Fanuc TP program (LS listing): 190220_hosenrohr_oV1.ls

/PROG  190220_hosenrohr_oV1
/ATTR
COMMENT	= "19-02-22 10:03:29";
PROG_SIZE	= 0;
DEFAULT_GROUP	= 1, 1, *, *, *;
/APPL
    ARC Welding Equipment: 1, *, *, *, *;
/MN
   1:  CALL HOME_ALL;
   1:  UFRAME_NUM = 1;
   1:  UTOOL_NUM = 3;
   1:  COL GUARD ADJUST 150;
   1:  ! -- Layer/Ebene 27 -- !;
   1:  PR[91] = PR[90];
   1:  PR[GP1:91,1] = PR[GP1:90,1] + -0.402;
   1:  PR[GP1:91,2] = PR[GP1:90,2] + 1.190;
   1:  PR[GP1:91,3] = PR[GP1:90,3] + 16.775;
   1:  !Sicherheitspunkt!;
   1:  PR[92] = PR[91];
   1:  PR[92] = PR[GP1:92,3] + 50;
   1:J PR[92];
   1:  !Schweissanfang anfahren!;
   1:L PR[91] R[100]mm/sec CNT100;
   1:  CALL LASER_DRAHT_START;
   1:  PR[GP1:91,1] = PR[GP1:90,1] + -0.660;
   1:  PR[GP1:91,2] = PR[GP1:90,2] + 1.301;
   1:L PR[91] R[100]mm/sec CNT100;
   1:  PR[GP1:91,1] = PR[GP1:90,1] + -2.989;
   1:  PR[GP1:91,2] = PR[GP1:90,2] + 2.142;
   1:L PR[91] R[100]mm/sec CNT100;
   1:  PR[GP1:91,1] = PR[GP1:90,1] + -5.273;
   1:  PR[GP1:91,2] = PR[GP1:90,2] + 6.132;
   1:L PR[91] R[100]mm/sec CNT100;
   1:  PR[GP1:91,1] = PR[GP1:90,1] + -8.308;
   1:  PR[GP1:91,2] = PR[GP1:90,2] + 15.071;
   1:L PR[91] R[100]mm/sec CNT100;
   1:  PR[GP1:91,1] = PR[GP1:90,1] + -9.096;
   1:  PR[GP1:91,2] = PR[GP1:90,2] + 16.647;
   1:L PR[91] R[100]mm/sec CNT100;
   1:  PR[GP1:91,1] = PR[GP1:90,1] + -15.340;
   1:  PR[GP1:91,2] = PR[GP1:90,2] + 24.664;
   1:L PR[91] R[100]mm/sec CNT100;
   1:  PR[GP1:91,1] = PR[GP1:90,1] + -15.998;
   1:  PR[GP1:91,2] = PR[GP1:90,2] + 25.324;
   1:L PR[91] R[100]mm/sec CNT100;
   1:  PR[GP1:91,1] = PR[GP1:90,1] + -25.382;
   1:  PR[GP1:91,2] = PR[GP1:90,2] + 31.412;
   1:L PR[91] R[100]mm/sec CNT100;
   1:  PR[GP1:91,1] = PR[GP1:90,1] + -36.399;
   1:  PR[GP1:91,2] = PR[GP1:90,2] + 34.262;
   1:L PR[91] R[100]mm/sec CNT100;
   1:  PR[GP1:91,1] = PR[GP1:90,1] + -36.821;
   1:  PR[GP1:91,2] = PR[GP1:90,2] + 34.270;
   1:L PR[91] R[100]mm/sec CNT100;
   1:  PR[GP1:91,1] = PR[GP1:90,1] + -47.006;
   1:  PR[GP1:91,2] = PR[GP1:90,2] + 33.504;
   1:L PR[91] R[100]mm/sec CNT100;
   1:  PR[GP1:91,1] = PR[GP1:90,1] + -47.901;
   1:  PR[GP1:91,2] = PR[GP1:90,2] + 33.351;
   1:L PR[91] R[100]mm/sec CNT100;
   1:  PR[GP1:91,1] = PR[GP1:90,1] + -48.764;
   1:  PR[GP1:91,2] = PR[GP1:90,2] + 33.031;
   1:L PR[91] R[100]mm/sec CNT100;
   1:  PR[GP1:91,1] = PR[GP1:90,1] + -57.526;
   1:  PR[GP1:91,2] = PR[GP1:90,2] + 29.256;
   1:L PR[91] R[100]mm/sec CNT100;
   1:  PR[GP1:91,1] = PR[GP1:90,1] + -58.611;
   1:  PR[GP1:91,2] = PR[GP1:90,2] + 28.601;
   1:L PR[91] R[100]mm/sec CNT100;
   1:  PR[GP1:91,1] = PR[GP1:90,1] + -59.584;
   1:  PR[GP1:91,2] = PR[GP1:90,2] + 27.731;
   1:L PR[91] R[100]mm/sec CNT100;
   1:  PR[GP1:91,1] = PR[GP1:90,1] + -66.238;
   1:  PR[GP1:91,2] = PR[GP1:90,2] + 21.668;
   1:L PR[91] R[100]mm/sec CNT100;
   1:  PR[GP1:91,1] = PR[GP1:90,1] + -67.162;
   1:  PR[GP1:91,2] = PR[GP1:90,2] + 20.463;
   1:L PR[91] R[100]mm/sec CNT100;
   1:  PR[GP1:91,1] = PR[GP1:90,1] + -67.875;
   1:  PR[GP1:91,2] = PR[GP1:90,2] + 19.051;
   1:L PR[91] R[100]mm/sec CNT100;
   1:  PR[GP1:91,1] = PR[GP1:90,1] + -71.993;
   1:  PR[GP1:91,2] = PR[GP1:90,2] + 11.491;
   1:L PR[91] R[100]mm/sec CNT100;
   1:  PR[GP1:91,1] = PR[GP1:90,1] + -72.454;
   1:  PR[GP1:91,2] = PR[GP1:90,2] + 9.892;
   1:L PR[91] R[100]mm/sec CNT100;
   1:  PR[GP1:91,1] = PR[GP1:90,1] + -72.617;
   1:  PR[GP1:91,2] = PR[GP1:90,2] + 8.149;
   1:L PR[91] R[100]mm/sec CNT100;
   1:  PR[GP1:91,1] = PR[GP1:90,1] + -73.992;
   1:  PR[GP1:91,2] = PR[GP1:90,2] + -0.094;
   1:L PR[91] R[100]mm/sec CNT100;
   1:  PR[GP1:91,1] = PR[GP1:90,1] + -73.819;
   1:  PR[GP1:91,2] = PR[GP1:90,2] + -1.941;
   1:L PR[91] R[100]mm/sec CNT100;
   1:  PR[GP1:91,1] = PR[GP1:90,1] + -72.460;
   1:  PR[GP1:91,2] = PR[GP1:90,2] + -10.015;
   1:L PR[91] R[100]mm/sec CNT100;
   1:  PR[GP1:91,1] = PR[GP1:90,1] + -71.991;
   1:  PR[GP1:91,2] = PR[GP1:90,2] + -11.644;
   1:L PR[91] R[100]mm/sec CNT100;
   1:  PR[GP1:91,1] = PR[GP1:90,1] + -71.216;
   1:  PR[GP1:91,2] = PR[GP1:90,2] + -13.179;
   1:L PR[91] R[100]mm/sec CNT100;
   1:  PR[GP1:91,1] = PR[GP1:90,1] + -67.168;
   1:  PR[GP1:91,2] = PR[GP1:90,2] + -20.599;
   1:L PR[91] R[100]mm/sec CNT100;
   1:  PR[GP1:91,1] = PR[GP1:90,1] + -66.239;
   1:  PR[GP1:91,2] = PR[GP1:90,2] + -21.810;
   1:L PR[91] R[100]mm/sec CNT100;
   1:  PR[GP1:91,1] = PR[GP1:90,1] + -65.065;
   1:  PR[GP1:91,2] = PR[GP1:90,2] + -22.860;
   1:L PR[91] R[100]mm/sec CNT100;
   1:  PR[GP1:91,1] = PR[GP1:90,1] + -58.609;
   1:  PR[GP1:91,2] = PR[GP1:90,2] + -28.747;
   1:L PR[91] R[100]mm/sec CNT100;
   1:  PR[GP1:91,1] = PR[GP1:90,1] + -57.539;
   1:  PR[GP1:91,2] = PR[GP1:90,2] + -29.392;
   1:L PR[91] R[100]mm/sec CNT100;
   1:  PR[GP1:91,1] = PR[GP1:90,1] + -56.298;
   1:  PR[GP1:91,2] = PR[GP1:90,2] + -29.853;
   1:L PR[91] R[100]mm/sec CNT100;
   1:  PR[GP1:91,1] = PR[GP1:90,1] + -47.885;
   1:  PR[GP1:91,2] = PR[GP1:90,2] + -33.498;
   1:L PR[91] R[100]mm/sec CNT100;
   1:  PR[GP1:91,1] = PR[GP1:90,1] + -47.006;
   1:  PR[GP1:91,2] = PR[GP1:90,2] + -33.648;
   1:L PR[91] R[100]mm/sec CNT100;
   1:  PR[GP1:91,1] = PR[GP1:90,1] + -36.821;
   1:  PR[GP1:91,2] = PR[GP1:90,2] + -34.414;
   1:L PR[91] R[100]mm/sec CNT100;
   1:  PR[GP1:91,1] = PR[GP1:90,1] + -36.385;
   1:  PR[GP1:91,2] = PR[GP1:90,2] + -34.406;
   1:L PR[91] R[100]mm/sec CNT100;
   1:  PR[GP1:91,1] = PR[GP1:90,1] + -35.945;
   1:  PR[GP1:91,2] = PR[GP1:90,2] + -34.315;
   1:L PR[91] R[100]mm/sec CNT100;
   1:  PR[GP1:91,1] = PR[GP1:90,1] + -25.382;
   1:  PR[GP1:91,2] = PR[GP1:90,2] + -31.557;
   1:L PR[91] R[100]mm/sec CNT100;
   1:  PR[GP1:91,1] = PR[GP1:90,1] + -15.998;
   1:  PR[GP1:91,2] = PR[GP1:90,2] + -25.468;
   1:L PR[91] R[100]mm/sec CNT100;
   1:  PR[GP1:91,1] = PR[GP1:90,1] + -15.340;
   1:  PR[GP1:91,2] = PR[GP1:90,2] + -24.808;
   1:L PR[91] R[100]mm/sec CNT100;
   1:  PR[GP1:91,1] = PR[GP1:90,1] + -9.096;
   1:  PR[GP1:91,2] = PR[GP1:90,2] + -16.791;
   1:L PR[91] R[100]mm/sec CNT100;
   1:  PR[GP1:91,1] = PR[GP1:90,1] + -8.309;
   1:  PR[GP1:91,2] = PR[GP1:90,2] + -15.219;
   1:L PR[91] R[100]mm/sec CNT100;
   1:  PR[GP1:91,1] = PR[GP1:90,1] + -5.290;
   1:  PR[GP1:91,2] = PR[GP1:90,2] + -6.326;
   1:L PR[91] R[100]mm/sec CNT100;
   1:  PR[GP1:91,1] = PR[GP1:90,1] + -4.379;
   1:  PR[GP1:91,2] = PR[GP1:90,2] + -3.772;
   1:L PR[91] R[100]mm/sec CNT100;
   1:  PR[GP1:91,1] = PR[GP1:90,1] + -3.822;
   1:  PR[GP1:91,2] = PR[GP1:90,2] + -3.156;
   1:L PR[91] R[100]mm/sec CNT100;
   1:  PR[GP1:91,1] = PR[GP1:90,1] + -3.023;
   1:  PR[GP1:91,2] = PR[GP1:90,2] + -2.452;
   1:L PR[91] R[100]mm/sec CNT100;
   1:  PR[GP1:91,1] = PR[GP1:90,1] + -2.740;
   1:  PR[GP1:91,2] = PR[GP1:90,2] + -2.161;
   1:L PR[91] R[100]mm/sec CNT100;
   1:  PR[GP1:91,1] = PR[GP1:90,1] + -2.333;
   1:  PR[GP1:91,2] = PR[GP1:90,2] + -1.998;
   1:L PR[91] R[100]mm/sec CNT100;
   1:  PR[GP1:91,1] = PR[GP1:90,1] + -0.802;
   1:  PR[GP1:91,2] = PR[GP1:90,2] + -1.217;
   1:L PR[91] R[100]mm/sec CNT100;
   1:  PR[GP1:91,1] = PR[GP1:90,1] + 0.616;
   1:  PR[GP1:91,2] = PR[GP1:90,2] + -1.334;
   1:L PR[91] R[100]mm/sec CNT100;
   1:  PR[GP1:91,1] = PR[GP1:90,1] + 0.873;
   1:  PR[GP1:91,2] = PR[GP1:90,2] + -1.445;
   1:L PR[91] R[100]mm/sec CNT100;
   1:  PR[GP1:91,1] = PR[GP1:90,1] + 3.204;
   1:  PR[GP1:91,2] = PR[GP1:90,2] + -2.287;
   1:L PR[91] R[100]mm/sec CNT100;
   1:  PR[GP1:91,1] = PR[GP1:90,1] + 3.775;
   1:  PR[GP1:91,2] = PR[GP1:90,2] + -3.292;
   1:L PR[91] R[100]mm/sec CNT100;
   1:  PR[GP1:91,1] = PR[GP1:90,1] + 5.076;
   1:  PR[GP1:91,2] = PR[GP1:90,2] + -5.769;
   1:L PR[91] R[100]mm/sec CNT100;
   1:  PR[GP1:91,1] = PR[GP1:90,1] + 5.465;
   1:  PR[GP1:91,2] = PR[GP1:90,2] + -6.220;
   1:L PR[91] R[100]mm/sec CNT100;
   1:  PR[GP1:91,1] = PR[GP1:90,1] + 8.520;
   1:  PR[GP1:91,2] = PR[GP1:90,2] + -15.214;
   1:L PR[91] R[100]mm/sec CNT100;
   1:  PR[GP1:91,1] = PR[GP1:90,1] + 9.306;
   1:  PR[GP1:91,2] = PR[GP1:90,2] + -16.783;
   1:L PR[91] R[100]mm/sec CNT100;
   1:  PR[GP1:91,1] = PR[GP1:90,1] + 15.550;
   1:  PR[GP1:91,2] = PR[GP1:90,2] + -24.804;
   1:L PR[91] R[100]mm/sec CNT100;
   1:  PR[GP1:91,1] = PR[GP1:90,1] + 16.209;
   1:  PR[GP1:91,2] = PR[GP1:90,2] + -25.466;
   1:L PR[91] R[100]mm/sec CNT100;
   1:  PR[GP1:91,1] = PR[GP1:90,1] + 25.593;
   1:  PR[GP1:91,2] = PR[GP1:90,2] + -31.555;
   1:L PR[91] R[100]mm/sec CNT100;
   1:  PR[GP1:91,1] = PR[GP1:90,1] + 36.611;
   1:  PR[GP1:91,2] = PR[GP1:90,2] + -34.406;
   1:L PR[91] R[100]mm/sec CNT100;
   1:  PR[GP1:91,1] = PR[GP1:90,1] + 37.032;
   1:  PR[GP1:91,2] = PR[GP1:90,2] + -34.414;
   1:L PR[91] R[100]mm/sec CNT100;
   1:  PR[GP1:91,1] = PR[GP1:90,1] + 47.218;
   1:  PR[GP1:91,2] = PR[GP1:90,2] + -33.648;
   1:L PR[91] R[100]mm/sec CNT100;
   1:  PR[GP1:91,1] = PR[GP1:90,1] + 48.113;
   1:  PR[GP1:91,2] = PR[GP1:90,2] + -33.495;
   1:L PR[91] R[100]mm/sec CNT100;
   1:  PR[GP1:91,1] = PR[GP1:90,1] + 48.975;
   1:  PR[GP1:91,2] = PR[GP1:90,2] + -33.175;
   1:L PR[91] R[100]mm/sec CNT100;
   1:  PR[GP1:91,1] = PR[GP1:90,1] + 57.738;
   1:  PR[GP1:91,2] = PR[GP1:90,2] + -29.401;
   1:L PR[91] R[100]mm/sec CNT100;
   1:  PR[GP1:91,1] = PR[GP1:90,1] + 58.824;
   1:  PR[GP1:91,2] = PR[GP1:90,2] + -28.746;
   1:L PR[91] R[100]mm/sec CNT100;
   1:  PR[GP1:91,1] = PR[GP1:90,1] + 59.797;
   1:  PR[GP1:91,2] = PR[GP1:90,2] + -27.876;
   1:L PR[91] R[100]mm/sec CNT100;
   1:  PR[GP1:91,1] = PR[GP1:90,1] + 66.450;
   1:  PR[GP1:91,2] = PR[GP1:90,2] + -21.811;
   1:L PR[91] R[100]mm/sec CNT100;
   1:  PR[GP1:91,1] = PR[GP1:90,1] + 67.375;
   1:  PR[GP1:91,2] = PR[GP1:90,2] + -20.606;
   1:L PR[91] R[100]mm/sec CNT100;
   1:  PR[GP1:91,1] = PR[GP1:90,1] + 68.088;
   1:  PR[GP1:91,2] = PR[GP1:90,2] + -19.193;
   1:L PR[91] R[100]mm/sec CNT100;
   1:  PR[GP1:91,1] = PR[GP1:90,1] + 72.207;
   1:  PR[GP1:91,2] = PR[GP1:90,2] + -11.638;
   1:L PR[91] R[100]mm/sec CNT100;
   1:  PR[GP1:91,1] = PR[GP1:90,1] + 72.667;
   1:  PR[GP1:91,2] = PR[GP1:90,2] + -10.040;
   1:L PR[91] R[100]mm/sec CNT100;
   1:  PR[GP1:91,1] = PR[GP1:90,1] + 72.830;
   1:  PR[GP1:91,2] = PR[GP1:90,2] + -8.297;
   1:L PR[91] R[100]mm/sec CNT100;
   1:  PR[GP1:91,1] = PR[GP1:90,1] + 74.205;
   1:  PR[GP1:91,2] = PR[GP1:90,2] + -0.050;
   1:L PR[91] R[100]mm/sec CNT100;
   1:  PR[GP1:91,1] = PR[GP1:90,1] + 74.032;
   1:  PR[GP1:91,2] = PR[GP1:90,2] + 1.797;
   1:L PR[91] R[100]mm/sec CNT100;
   1:  PR[GP1:91,1] = PR[GP1:90,1] + 72.673;
   1:  PR[GP1:91,2] = PR[GP1:90,2] + 9.874;
   1:L PR[91] R[100]mm/sec CNT100;
   1:  PR[GP1:91,1] = PR[GP1:90,1] + 72.204;
   1:  PR[GP1:91,2] = PR[GP1:90,2] + 11.504;
   1:L PR[91] R[100]mm/sec CNT100;
   1:  PR[GP1:91,1] = PR[GP1:90,1] + 71.429;
   1:  PR[GP1:91,2] = PR[GP1:90,2] + 13.039;
   1:L PR[91] R[100]mm/sec CNT100;
   1:  PR[GP1:91,1] = PR[GP1:90,1] + 67.381;
   1:  PR[GP1:91,2] = PR[GP1:90,2] + 20.454;
   1:L PR[91] R[100]mm/sec CNT100;
   1:  PR[GP1:91,1] = PR[GP1:90,1] + 66.452;
   1:  PR[GP1:91,2] = PR[GP1:90,2] + 21.665;
   1:L PR[91] R[100]mm/sec CNT100;
   1:  PR[GP1:91,1] = PR[GP1:90,1] + 65.278;
   1:  PR[GP1:91,2] = PR[GP1:90,2] + 22.715;
   1:L PR[91] R[100]mm/sec CNT100;
   1:  PR[GP1:91,1] = PR[GP1:90,1] + 58.821;
   1:  PR[GP1:91,2] = PR[GP1:90,2] + 28.604;
   1:L PR[91] R[100]mm/sec CNT100;
   1:  PR[GP1:91,1] = PR[GP1:90,1] + 57.752;
   1:  PR[GP1:91,2] = PR[GP1:90,2] + 29.249;
   1:L PR[91] R[100]mm/sec CNT100;
   1:  PR[GP1:91,1] = PR[GP1:90,1] + 56.510;
   1:  PR[GP1:91,2] = PR[GP1:90,2] + 29.710;
   1:L PR[91] R[100]mm/sec CNT100;
   1:  PR[GP1:91,1] = PR[GP1:90,1] + 48.097;
   1:  PR[GP1:91,2] = PR[GP1:90,2] + 33.354;
   1:L PR[91] R[100]mm/sec CNT100;
   1:  PR[GP1:91,1] = PR[GP1:90,1] + 47.218;
   1:  PR[GP1:91,2] = PR[GP1:90,2] + 33.504;
   1:L PR[91] R[100]mm/sec CNT100;
   1:  PR[GP1:91,1] = PR[GP1:90,1] + 37.032;
   1:  PR[GP1:91,2] = PR[GP1:90,2] + 34.270;
   1:L PR[91] R[100]mm/sec CNT100;
   1:  PR[GP1:91,1] = PR[GP1:90,1] + 36.596;
   1:  PR[GP1:91,2] = PR[GP1:90,2] + 34.262;
   1:L PR[91] R[100]mm/sec CNT100;
   1:  PR[GP1:91,1] = PR[GP1:90,1] + 36.157;
   1:  PR[GP1:91,2] = PR[GP1:90,2] + 34.171;
   1:L PR[91] R[100]mm/sec CNT100;
   1:  PR[GP1:91,1] = PR[GP1:90,1] + 25.593;
   1:  PR[GP1:91,2] = PR[GP1:90,2] + 31.412;
   1:L PR[91] R[100]mm/sec CNT100;
   1:  PR[GP1:91,1] = PR[GP1:90,1] + 16.209;
   1:  PR[GP1:91,2] = PR[GP1:90,2] + 25.322;
   1:L PR[91] R[100]mm/sec CNT100;
   1:  PR[GP1:91,1] = PR[GP1:90,1] + 15.550;
   1:  PR[GP1:91,2] = PR[GP1:90,2] + 24.660;
   1:L PR[91] R[100]mm/sec CNT100;
   1:  PR[GP1:91,1] = PR[GP1:90,1] + 9.306;
   1:  PR[GP1:91,2] = PR[GP1:90,2] + 16.639;
   1:L PR[91] R[100]mm/sec CNT100;
   1:  PR[GP1:91,1] = PR[GP1:90,1] + 8.518;
   1:  PR[GP1:91,2] = PR[GP1:90,2] + 15.066;
   1:L PR[91] R[100]mm/sec CNT100;
   1:  PR[GP1:91,1] = PR[GP1:90,1] + 5.502;
   1:  PR[GP1:91,2] = PR[GP1:90,2] + 6.182;
   1:L PR[91] R[100]mm/sec CNT100;
   1:  PR[GP1:91,1] = PR[GP1:90,1] + 4.592;
   1:  PR[GP1:91,2] = PR[GP1:90,2] + 3.627;
   1:L PR[91] R[100]mm/sec CNT100;
   1:  PR[GP1:91,1] = PR[GP1:90,1] + 4.036;
   1:  PR[GP1:91,2] = PR[GP1:90,2] + 3.013;
   1:L PR[91] R[100]mm/sec CNT100;
   1:  PR[GP1:91,1] = PR[GP1:90,1] + 3.236;
   1:  PR[GP1:91,2] = PR[GP1:90,2] + 2.309;
   1:L PR[91] R[100]mm/sec CNT100;
   1:  PR[GP1:91,1] = PR[GP1:90,1] + 2.954;
   1:  PR[GP1:91,2] = PR[GP1:90,2] + 2.018;
   1:L PR[91] R[100]mm/sec CNT100;
   1:  PR[GP1:91,1] = PR[GP1:90,1] + 2.547;
   1:  PR[GP1:91,2] = PR[GP1:90,2] + 1.854;
   1:L PR[91] R[100]mm/sec CNT100;
   1:  PR[GP1:91,1] = PR[GP1:90,1] + 1.015;
   1:  PR[GP1:91,2] = PR[GP1:90,2] + 1.073;
   1:L PR[91] R[100]mm/sec CNT100;
   1:  ! -- Layer/Ebene 28 -- !;
   1:  PR[91] = PR[90];
   1:  PR[GP1:91,1] = PR[GP1:90,1] + -1.935;
   1:  PR[GP1:91,2] = PR[GP1:90,2] + 1.929;
   1:  PR[GP1:91,3] = PR[GP1:90,3] + 17.385;
   1:L PR[91] R[100]mm/sec CNT100;
   1:  PR[GP1:91,1] = PR[GP1:90,1] + -2.796;
   1:  PR[GP1:91,2] = PR[GP1:90,2] + 2.294;
   1:L PR[91] R[100]mm/sec CNT100;
   1:  PR[GP1:91,1] = PR[GP1:90,1] + -5.248;
   1:  PR[GP1:91,2] = PR[GP1:90,2] + 6.572;
   1:L PR[91] R[100]mm/sec CNT100;
   1:  PR[GP1:91,1] = PR[GP1:90,1] + -7.950;
   1:  PR[GP1:91,2] = PR[GP1:90,2] + 14.528;
   1:L PR[91] R[100]mm/sec CNT100;
   1:  PR[GP1:91,1] = PR[GP1:90,1] + -9.175;
   1:  PR[GP1:91,2] = PR[GP1:90,2] + 16.979;
   1:L PR[91] R[100]mm/sec CNT100;
   1:  PR[GP1:91,1] = PR[GP1:90,1] + -14.817;
   1:  PR[GP1:91,2] = PR[GP1:90,2] + 24.222;
   1:L PR[91] R[100]mm/sec CNT100;
   1:  PR[GP1:91,1] = PR[GP1:90,1] + -16.126;
   1:  PR[GP1:91,2] = PR[GP1:90,2] + 25.535;
   1:L PR[91] R[100]mm/sec CNT100;
   1:  PR[GP1:91,1] = PR[GP1:90,1] + -24.751;
   1:  PR[GP1:91,2] = PR[GP1:90,2] + 31.136;
   1:L PR[91] R[100]mm/sec CNT100;
   1:  PR[GP1:91,1] = PR[GP1:90,1] + -25.479;
   1:  PR[GP1:91,2] = PR[GP1:90,2] + 31.508;
   1:L PR[91] R[100]mm/sec CNT100;
   1:  PR[GP1:91,1] = PR[GP1:90,1] + -34.683;
   1:  PR[GP1:91,2] = PR[GP1:90,2] + 33.823;
   1:L PR[91] R[100]mm/sec CNT100;
   1:  PR[GP1:91,1] = PR[GP1:90,1] + -36.395;
   1:  PR[GP1:91,2] = PR[GP1:90,2] + 34.266;
   1:L PR[91] R[100]mm/sec CNT100;
   1:  PR[GP1:91,1] = PR[GP1:90,1] + -47.334;
   1:  PR[GP1:91,2] = PR[GP1:90,2] + 33.451;
   1:L PR[91] R[100]mm/sec CNT100;
   1:  PR[GP1:91,1] = PR[GP1:90,1] + -47.835;
   1:  PR[GP1:91,2] = PR[GP1:90,2] + 33.366;
   1:L PR[91] R[100]mm/sec CNT100;
   1:  PR[GP1:91,1] = PR[GP1:90,1] + -48.324;
   1:  PR[GP1:91,2] = PR[GP1:90,2] + 33.184;
   1:L PR[91] R[100]mm/sec CNT100;
   1:  PR[GP1:91,1] = PR[GP1:90,1] + -57.721;
   1:  PR[GP1:91,2] = PR[GP1:90,2] + 29.136;
   1:L PR[91] R[100]mm/sec CNT100;
   1:  PR[GP1:91,1] = PR[GP1:90,1] + -58.486;
   1:  PR[GP1:91,2] = PR[GP1:90,2] + 28.675;
   1:L PR[91] R[100]mm/sec CNT100;
   1:  PR[GP1:91,1] = PR[GP1:90,1] + -66.319;
   1:  PR[GP1:91,2] = PR[GP1:90,2] + 21.549;
   1:L PR[91] R[100]mm/sec CNT100;
   1:  PR[GP1:91,1] = PR[GP1:90,1] + -67.028;
   1:  PR[GP1:91,2] = PR[GP1:90,2] + 20.624;
   1:L PR[91] R[100]mm/sec CNT100;
   1:  PR[GP1:91,1] = PR[GP1:90,1] + -67.582;
   1:  PR[GP1:91,2] = PR[GP1:90,2] + 19.527;
   1:L PR[91] R[100]mm/sec CNT100;
   1:  PR[GP1:91,1] = PR[GP1:90,1] + -71.999;
   1:  PR[GP1:91,2] = PR[GP1:90,2] + 11.419;
   1:L PR[91] R[100]mm/sec CNT100;
   1:  PR[GP1:91,1] = PR[GP1:90,1] + -72.365;
   1:  PR[GP1:91,2] = PR[GP1:90,2] + 10.149;
   1:L PR[91] R[100]mm/sec CNT100;
   1:  PR[GP1:91,1] = PR[GP1:90,1] + -72.496;
   1:  PR[GP1:91,2] = PR[GP1:90,2] + 8.747;
   1:L PR[91] R[100]mm/sec CNT100;
   1:  PR[GP1:91,1] = PR[GP1:90,1] + -73.971;
   1:  PR[GP1:91,2] = PR[GP1:90,2] + -0.094;
   1:L PR[91] R[100]mm/sec CNT100;
   1:  PR[GP1:91,1] = PR[GP1:90,1] + -73.828;
   1:  PR[GP1:91,2] = PR[GP1:90,2] + -1.613;
   1:L PR[91] R[100]mm/sec CNT100;
   1:  PR[GP1:91,1] = PR[GP1:90,1] + -72.371;
   1:  PR[GP1:91,2] = PR[GP1:90,2] + -10.272;
   1:L PR[91] R[100]mm/sec CNT100;
   1:  PR[GP1:91,1] = PR[GP1:90,1] + -71.996;
   1:  PR[GP1:91,2] = PR[GP1:90,2] + -11.573;
   1:L PR[91] R[100]mm/sec CNT100;
   1:  PR[GP1:91,1] = PR[GP1:90,1] + -71.375;
   1:  PR[GP1:91,2] = PR[GP1:90,2] + -12.803;
   1:L PR[91] R[100]mm/sec CNT100;
   1:  PR[GP1:91,1] = PR[GP1:90,1] + -67.034;
   1:  PR[GP1:91,2] = PR[GP1:90,2] + -20.761;
   1:L PR[91] R[100]mm/sec CNT100;
   1:  PR[GP1:91,1] = PR[GP1:90,1] + -66.320;
   1:  PR[GP1:91,2] = PR[GP1:90,2] + -21.691;
   1:L PR[91] R[100]mm/sec CNT100;
   1:  PR[GP1:91,1] = PR[GP1:90,1] + -65.409;
   1:  PR[GP1:91,2] = PR[GP1:90,2] + -22.506;
   1:L PR[91] R[100]mm/sec CNT100;
   1:  PR[GP1:91,1] = PR[GP1:90,1] + -58.485;
   1:  PR[GP1:91,2] = PR[GP1:90,2] + -28.819;
   1:L PR[91] R[100]mm/sec CNT100;
   1:  PR[GP1:91,1] = PR[GP1:90,1] + -57.734;
   1:  PR[GP1:91,2] = PR[GP1:90,2] + -29.272;
   1:L PR[91] R[100]mm/sec CNT100;
   1:  PR[GP1:91,1] = PR[GP1:90,1] + -56.842;
   1:  PR[GP1:91,2] = PR[GP1:90,2] + -29.603;
   1:L PR[91] R[100]mm/sec CNT100;
   1:  PR[GP1:91,1] = PR[GP1:90,1] + -47.819;
   1:  PR[GP1:91,2] = PR[GP1:90,2] + -33.512;
   1:L PR[91] R[100]mm/sec CNT100;
   1:  PR[GP1:91,1] = PR[GP1:90,1] + -47.334;
   1:  PR[GP1:91,2] = PR[GP1:90,2] + -33.595;
   1:L PR[91] R[100]mm/sec CNT100;
   1:  PR[GP1:91,1] = PR[GP1:90,1] + -36.395;
   1:  PR[GP1:91,2] = PR[GP1:90,2] + -34.410;
   1:L PR[91] R[100]mm/sec CNT100;
   1:  PR[GP1:91,1] = PR[GP1:90,1] + -34.683;
   1:  PR[GP1:91,2] = PR[GP1:90,2] + -33.967;
   1:L PR[91] R[100]mm/sec CNT100;
   1:  PR[GP1:91,1] = PR[GP1:90,1] + -25.479;
   1:  PR[GP1:91,2] = PR[GP1:90,2] + -31.652;
   1:L PR[91] R[100]mm/sec CNT100;
   1:  PR[GP1:91,1] = PR[GP1:90,1] + -24.751;
   1:  PR[GP1:91,2] = PR[GP1:90,2] + -31.280;
   1:L PR[91] R[100]mm/sec CNT100;
   1:  PR[GP1:91,1] = PR[GP1:90,1] + -16.126;
   1:  PR[GP1:91,2] = PR[GP1:90,2] + -25.679;
   1:L PR[91] R[100]mm/sec CNT100;
   1:  PR[GP1:91,1] = PR[GP1:90,1] + -14.817;
   1:  PR[GP1:91,2] = PR[GP1:90,2] + -24.366;
   1:L PR[91] R[100]mm/sec CNT100;
   1:  PR[GP1:91,1] = PR[GP1:90,1] + -9.175;
   1:  PR[GP1:91,2] = PR[GP1:90,2] + -17.123;
   1:L PR[91] R[100]mm/sec CNT100;
   1:  PR[GP1:91,1] = PR[GP1:90,1] + -7.951;
   1:  PR[GP1:91,2] = PR[GP1:90,2] + -14.678;
   1:L PR[91] R[100]mm/sec CNT100;
   1:  PR[GP1:91,1] = PR[GP1:90,1] + -5.266;
   1:  PR[GP1:91,2] = PR[GP1:90,2] + -6.766;
   1:L PR[91] R[100]mm/sec CNT100;
   1:  PR[GP1:91,1] = PR[GP1:90,1] + -4.413;
   1:  PR[GP1:91,2] = PR[GP1:90,2] + -4.372;
   1:L PR[91] R[100]mm/sec CNT100;
   1:  PR[GP1:91,1] = PR[GP1:90,1] + -2.724;
   1:  PR[GP1:91,2] = PR[GP1:90,2] + -2.505;
   1:L PR[91] R[100]mm/sec CNT100;
   1:  PR[GP1:91,1] = PR[GP1:90,1] + -2.463;
   1:  PR[GP1:91,2] = PR[GP1:90,2] + -2.267;
   1:L PR[91] R[100]mm/sec CNT100;
   1:  PR[GP1:91,1] = PR[GP1:90,1] + -1.968;
   1:  PR[GP1:91,2] = PR[GP1:90,2] + -2.068;
   1:L PR[91] R[100]mm/sec CNT100;
   1:  PR[GP1:91,1] = PR[GP1:90,1] + -1.406;
   1:  PR[GP1:91,2] = PR[GP1:90,2] + -1.781;
   1:L PR[91] R[100]mm/sec CNT100;
   1:  PR[GP1:91,1] = PR[GP1:90,1] + 2.147;
   1:  PR[GP1:91,2] = PR[GP1:90,2] + -2.073;
   1:L PR[91] R[100]mm/sec CNT100;
   1:  PR[GP1:91,1] = PR[GP1:90,1] + 3.020;
   1:  PR[GP1:91,2] = PR[GP1:90,2] + -2.443;
   1:L PR[91] R[100]mm/sec CNT100;
   1:  PR[GP1:91,1] = PR[GP1:90,1] + 4.920;
   1:  PR[GP1:91,2] = PR[GP1:90,2] + -6.058;
   1:L PR[91] R[100]mm/sec CNT100;
   1:  PR[GP1:91,1] = PR[GP1:90,1] + 5.441;
   1:  PR[GP1:91,2] = PR[GP1:90,2] + -6.659;
   1:L PR[91] R[100]mm/sec CNT100;
   1:  PR[GP1:91,1] = PR[GP1:90,1] + 8.162;
   1:  PR[GP1:91,2] = PR[GP1:90,2] + -14.673;
   1:L PR[91] R[100]mm/sec CNT100;
   1:  PR[GP1:91,1] = PR[GP1:90,1] + 9.385;
   1:  PR[GP1:91,2] = PR[GP1:90,2] + -17.113;
   1:L PR[91] R[100]mm/sec CNT100;
   1:  PR[GP1:91,1] = PR[GP1:90,1] + 15.027;
   1:  PR[GP1:91,2] = PR[GP1:90,2] + -24.361;
   1:L PR[91] R[100]mm/sec CNT100;
   1:  PR[GP1:91,1] = PR[GP1:90,1] + 16.336;
   1:  PR[GP1:91,2] = PR[GP1:90,2] + -25.677;
   1:L PR[91] R[100]mm/sec CNT100;
   1:  PR[GP1:91,1] = PR[GP1:90,1] + 24.961;
   1:  PR[GP1:91,2] = PR[GP1:90,2] + -31.278;
   1:L PR[91] R[100]mm/sec CNT100;
   1:  PR[GP1:91,1] = PR[GP1:90,1] + 25.689;
   1:  PR[GP1:91,2] = PR[GP1:90,2] + -31.650;
   1:L PR[91] R[100]mm/sec CNT100;
   1:  PR[GP1:91,1] = PR[GP1:90,1] + 34.896;
   1:  PR[GP1:91,2] = PR[GP1:90,2] + -33.967;
   1:L PR[91] R[100]mm/sec CNT100;
   1:  PR[GP1:91,1] = PR[GP1:90,1] + 36.607;
   1:  PR[GP1:91,2] = PR[GP1:90,2] + -34.410;
   1:L PR[91] R[100]mm/sec CNT100;
   1:  PR[GP1:91,1] = PR[GP1:90,1] + 47.546;
   1:  PR[GP1:91,2] = PR[GP1:90,2] + -33.595;
   1:L PR[91] R[100]mm/sec CNT100;
   1:  PR[GP1:91,1] = PR[GP1:90,1] + 48.047;
   1:  PR[GP1:91,2] = PR[GP1:90,2] + -33.510;
   1:L PR[91] R[100]mm/sec CNT100;
   1:  PR[GP1:91,1] = PR[GP1:90,1] + 48.536;
   1:  PR[GP1:91,2] = PR[GP1:90,2] + -33.328;
   1:L PR[91] R[100]mm/sec CNT100;
   1:  PR[GP1:91,1] = PR[GP1:90,1] + 57.934;
   1:  PR[GP1:91,2] = PR[GP1:90,2] + -29.281;
   1:L PR[91] R[100]mm/sec CNT100;
   1:  PR[GP1:91,1] = PR[GP1:90,1] + 58.698;
   1:  PR[GP1:91,2] = PR[GP1:90,2] + -28.820;
   1:L PR[91] R[100]mm/sec CNT100;
   1:  PR[GP1:91,1] = PR[GP1:90,1] + 66.532;
   1:  PR[GP1:91,2] = PR[GP1:90,2] + -21.692;
   1:L PR[91] R[100]mm/sec CNT100;
   1:  PR[GP1:91,1] = PR[GP1:90,1] + 67.241;
   1:  PR[GP1:91,2] = PR[GP1:90,2] + -20.767;
   1:L PR[91] R[100]mm/sec CNT100;
   1:  PR[GP1:91,1] = PR[GP1:90,1] + 67.795;
   1:  PR[GP1:91,2] = PR[GP1:90,2] + -19.670;
   1:L PR[91] R[100]mm/sec CNT100;
   1:  PR[GP1:91,1] = PR[GP1:90,1] + 72.212;
   1:  PR[GP1:91,2] = PR[GP1:90,2] + -11.567;
   1:L PR[91] R[100]mm/sec CNT100;
   1:  PR[GP1:91,1] = PR[GP1:90,1] + 72.578;
   1:  PR[GP1:91,2] = PR[GP1:90,2] + -10.297;
   1:L PR[91] R[100]mm/sec CNT100;
   1:  PR[GP1:91,1] = PR[GP1:90,1] + 72.709;
   1:  PR[GP1:91,2] = PR[GP1:90,2] + -8.894;
   1:L PR[91] R[100]mm/sec CNT100;
   1:  PR[GP1:91,1] = PR[GP1:90,1] + 74.184;
   1:  PR[GP1:91,2] = PR[GP1:90,2] + -0.050;
   1:L PR[91] R[100]mm/sec CNT100;
   1:  PR[GP1:91,1] = PR[GP1:90,1] + 74.042;
   1:  PR[GP1:91,2] = PR[GP1:90,2] + 1.469;
   1:L PR[91] R[100]mm/sec CNT100;
   1:  PR[GP1:91,1] = PR[GP1:90,1] + 72.584;
   1:  PR[GP1:91,2] = PR[GP1:90,2] + 10.132;
   1:L PR[91] R[100]mm/sec CNT100;
   1:  PR[GP1:91,1] = PR[GP1:90,1] + 72.209;
   1:  PR[GP1:91,2] = PR[GP1:90,2] + 11.432;
   1:L PR[91] R[100]mm/sec CNT100;
   1:  PR[GP1:91,1] = PR[GP1:90,1] + 71.589;
   1:  PR[GP1:91,2] = PR[GP1:90,2] + 12.662;
   1:L PR[91] R[100]mm/sec CNT100;
   1:  PR[GP1:91,1] = PR[GP1:90,1] + 67.247;
   1:  PR[GP1:91,2] = PR[GP1:90,2] + 20.615;
   1:L PR[91] R[100]mm/sec CNT100;
   1:  PR[GP1:91,1] = PR[GP1:90,1] + 66.533;
   1:  PR[GP1:91,2] = PR[GP1:90,2] + 21.546;
   1:L PR[91] R[100]mm/sec CNT100;
   1:  PR[GP1:91,1] = PR[GP1:90,1] + 65.622;
   1:  PR[GP1:91,2] = PR[GP1:90,2] + 22.361;
   1:L PR[91] R[100]mm/sec CNT100;
   1:  PR[GP1:91,1] = PR[GP1:90,1] + 58.698;
   1:  PR[GP1:91,2] = PR[GP1:90,2] + 28.676;
   1:L PR[91] R[100]mm/sec CNT100;
   1:  PR[GP1:91,1] = PR[GP1:90,1] + 57.947;
   1:  PR[GP1:91,2] = PR[GP1:90,2] + 29.129;
   1:L PR[91] R[100]mm/sec CNT100;
   1:  PR[GP1:91,1] = PR[GP1:90,1] + 57.055;
   1:  PR[GP1:91,2] = PR[GP1:90,2] + 29.461;
   1:L PR[91] R[100]mm/sec CNT100;
   1:  PR[GP1:91,1] = PR[GP1:90,1] + 48.031;
   1:  PR[GP1:91,2] = PR[GP1:90,2] + 33.368;
   1:L PR[91] R[100]mm/sec CNT100;
   1:  PR[GP1:91,1] = PR[GP1:90,1] + 47.546;
   1:  PR[GP1:91,2] = PR[GP1:90,2] + 33.451;
   1:L PR[91] R[100]mm/sec CNT100;
   1:  PR[GP1:91,1] = PR[GP1:90,1] + 36.650;
   1:  PR[GP1:91,2] = PR[GP1:90,2] + 34.271;
   1:L PR[91] R[100]mm/sec CNT100;
   1:  PR[GP1:91,1] = PR[GP1:90,1] + 36.577;
   1:  PR[GP1:91,2] = PR[GP1:90,2] + 34.263;
   1:L PR[91] R[100]mm/sec CNT100;
   1:  PR[GP1:91,1] = PR[GP1:90,1] + 34.897;
   1:  PR[GP1:91,2] = PR[GP1:90,2] + 33.823;
   1:L PR[91] R[100]mm/sec CNT100;
   1:  PR[GP1:91,1] = PR[GP1:90,1] + 25.689;
   1:  PR[GP1:91,2] = PR[GP1:90,2] + 31.506;
   1:L PR[91] R[100]mm/sec CNT100;
   1:  PR[GP1:91,1] = PR[GP1:90,1] + 24.961;
   1:  PR[GP1:91,2] = PR[GP1:90,2] + 31.134;
   1:L PR[91] R[100]mm/sec CNT100;
   1:  PR[GP1:91,1] = PR[GP1:90,1] + 16.336;
   1:  PR[GP1:91,2] = PR[GP1:90,2] + 25.533;
   1:L PR[91] R[100]mm/sec CNT100;
   1:  PR[GP1:91,1] = PR[GP1:90,1] + 15.027;
   1:  PR[GP1:91,2] = PR[GP1:90,2] + 24.217;
   1:L PR[91] R[100]mm/sec CNT100;
   1:  PR[GP1:91,1] = PR[GP1:90,1] + 9.385;
   1:  PR[GP1:91,2] = PR[GP1:90,2] + 16.969;
   1:L PR[91] R[100]mm/sec CNT100;
   1:  PR[GP1:91,1] = PR[GP1:90,1] + 8.160;
   1:  PR[GP1:91,2] = PR[GP1:90,2] + 14.523;
   1:L PR[91] R[100]mm/sec CNT100;
   1:  PR[GP1:91,1] = PR[GP1:90,1] + 5.477;
   1:  PR[GP1:91,2] = PR[GP1:90,2] + 6.622;
   1:L PR[91] R[100]mm/sec CNT100;
   1:  PR[GP1:91,1] = PR[GP1:90,1] + 4.629;
   1:  PR[GP1:91,2] = PR[GP1:90,2] + 4.238;
   1:L PR[91] R[100]mm/sec CNT100;
   1:  PR[GP1:91,1] = PR[GP1:90,1] + 4.333;
   1:  PR[GP1:91,2] = PR[GP1:90,2] + 3.880;
   1:L PR[91] R[100]mm/sec CNT100;
   1:  PR[GP1:91,1] = PR[GP1:90,1] + 2.936;
   1:  PR[GP1:91,2] = PR[GP1:90,2] + 2.360;
   1:L PR[91] R[100]mm/sec CNT100;
   1:  PR[GP1:91,1] = PR[GP1:90,1] + 2.677;
   1:  PR[GP1:91,2] = PR[GP1:90,2] + 2.124;
   1:L PR[91] R[100]mm/sec CNT100;
   1:  PR[GP1:91,1] = PR[GP1:90,1] + 2.182;
   1:  PR[GP1:91,2] = PR[GP1:90,2] + 1.924;
   1:L PR[91] R[100]mm/sec CNT100;
   1:  PR[GP1:91,1] = PR[GP1:90,1] + 1.619;
   1:  PR[GP1:91,2] = PR[GP1:90,2] + 1.638;
   1:L PR[91] R[100]mm/sec CNT100;
   1:  ! -- Layer/Ebene 29 -- !;
   1:  PR[91] = PR[90];
   1:  PR[GP1:91,1] = PR[GP1:90,1] + -2.280;
   1:  PR[GP1:91,2] = PR[GP1:90,2] + 2.492;
   1:  PR[GP1:91,3] = PR[GP1:90,3] + 17.995;
   1:L PR[91] R[100]mm/sec CNT100;
   1:  PR[GP1:91,1] = PR[GP1:90,1] + -2.743;
   1:  PR[GP1:91,2] = PR[GP1:90,2] + 2.817;
   1:L PR[91] R[100]mm/sec CNT100;
   1:  PR[GP1:91,1] = PR[GP1:90,1] + -3.008;
   1:  PR[GP1:91,2] = PR[GP1:90,2] + 3.141;
   1:L PR[91] R[100]mm/sec CNT100;
   1:  PR[GP1:91,1] = PR[GP1:90,1] + -5.224;
   1:  PR[GP1:91,2] = PR[GP1:90,2] + 7.012;
   1:L PR[91] R[100]mm/sec CNT100;
   1:  PR[GP1:91,1] = PR[GP1:90,1] + -7.592;
   1:  PR[GP1:91,2] = PR[GP1:90,2] + 13.985;
   1:L PR[91] R[100]mm/sec CNT100;
   1:  PR[GP1:91,1] = PR[GP1:90,1] + -9.255;
   1:  PR[GP1:91,2] = PR[GP1:90,2] + 17.310;
   1:L PR[91] R[100]mm/sec CNT100;
   1:  PR[GP1:91,1] = PR[GP1:90,1] + -14.295;
   1:  PR[GP1:91,2] = PR[GP1:90,2] + 23.781;
   1:L PR[91] R[100]mm/sec CNT100;
   1:  PR[GP1:91,1] = PR[GP1:90,1] + -16.254;
   1:  PR[GP1:91,2] = PR[GP1:90,2] + 25.746;
   1:L PR[91] R[100]mm/sec CNT100;
   1:  PR[GP1:91,1] = PR[GP1:90,1] + -24.101;
   1:  PR[GP1:91,2] = PR[GP1:90,2] + 30.842;
   1:L PR[91] R[100]mm/sec CNT100;
   1:  PR[GP1:91,1] = PR[GP1:90,1] + -25.608;
   1:  PR[GP1:91,2] = PR[GP1:90,2] + 31.612;
   1:L PR[91] R[100]mm/sec CNT100;
   1:  PR[GP1:91,1] = PR[GP1:90,1] + -35.900;
   1:  PR[GP1:91,2] = PR[GP1:90,2] + 34.201;
   1:L PR[91] R[100]mm/sec CNT100;
   1:  PR[GP1:91,1] = PR[GP1:90,1] + -36.449;
   1:  PR[GP1:91,2] = PR[GP1:90,2] + 34.290;
   1:L PR[91] R[100]mm/sec CNT100;
   1:  PR[GP1:91,1] = PR[GP1:90,1] + -43.478;
   1:  PR[GP1:91,2] = PR[GP1:90,2] + 33.713;
   1:L PR[91] R[100]mm/sec CNT100;
   1:  PR[GP1:91,1] = PR[GP1:90,1] + -47.662;
   1:  PR[GP1:91,2] = PR[GP1:90,2] + 33.399;
   1:L PR[91] R[100]mm/sec CNT100;
   1:  PR[GP1:91,1] = PR[GP1:90,1] + -47.770;
   1:  PR[GP1:91,2] = PR[GP1:90,2] + 33.380;
   1:L PR[91] R[100]mm/sec CNT100;
   1:  PR[GP1:91,1] = PR[GP1:90,1] + -47.884;
   1:  PR[GP1:91,2] = PR[GP1:90,2] + 33.338;
   1:L PR[91] R[100]mm/sec CNT100;
   1:  PR[GP1:91,1] = PR[GP1:90,1] + -57.916;
   1:  PR[GP1:91,2] = PR[GP1:90,2] + 29.016;
   1:L PR[91] R[100]mm/sec CNT100;
   1:  PR[GP1:91,1] = PR[GP1:90,1] + -58.362;
   1:  PR[GP1:91,2] = PR[GP1:90,2] + 28.747;
   1:L PR[91] R[100]mm/sec CNT100;
   1:  PR[GP1:91,1] = PR[GP1:90,1] + -66.400;
   1:  PR[GP1:91,2] = PR[GP1:90,2] + 21.430;
   1:L PR[91] R[100]mm/sec CNT100;
   1:  PR[GP1:91,1] = PR[GP1:90,1] + -66.894;
   1:  PR[GP1:91,2] = PR[GP1:90,2] + 20.786;
   1:L PR[91] R[100]mm/sec CNT100;
   1:  PR[GP1:91,1] = PR[GP1:90,1] + -67.289;
   1:  PR[GP1:91,2] = PR[GP1:90,2] + 20.004;
   1:L PR[91] R[100]mm/sec CNT100;
   1:  PR[GP1:91,1] = PR[GP1:90,1] + -72.004;
   1:  PR[GP1:91,2] = PR[GP1:90,2] + 11.348;
   1:L PR[91] R[100]mm/sec CNT100;
   1:  PR[GP1:91,1] = PR[GP1:90,1] + -72.275;
   1:  PR[GP1:91,2] = PR[GP1:90,2] + 10.407;
   1:L PR[91] R[100]mm/sec CNT100;
   1:  PR[GP1:91,1] = PR[GP1:90,1] + -72.375;
   1:  PR[GP1:91,2] = PR[GP1:90,2] + 9.344;
   1:L PR[91] R[100]mm/sec CNT100;
   1:  PR[GP1:91,1] = PR[GP1:90,1] + -73.949;
   1:  PR[GP1:91,2] = PR[GP1:90,2] + -0.094;
   1:L PR[91] R[100]mm/sec CNT100;
   1:  PR[GP1:91,1] = PR[GP1:90,1] + -73.838;
   1:  PR[GP1:91,2] = PR[GP1:90,2] + -1.285;
   1:L PR[91] R[100]mm/sec CNT100;
   1:  PR[GP1:91,1] = PR[GP1:90,1] + -72.282;
   1:  PR[GP1:91,2] = PR[GP1:90,2] + -10.529;
   1:L PR[91] R[100]mm/sec CNT100;
   1:  PR[GP1:91,1] = PR[GP1:90,1] + -72.002;
   1:  PR[GP1:91,2] = PR[GP1:90,2] + -11.501;
   1:L PR[91] R[100]mm/sec CNT100;
   1:  PR[GP1:91,1] = PR[GP1:90,1] + -71.535;
   1:  PR[GP1:91,2] = PR[GP1:90,2] + -12.426;
   1:L PR[91] R[100]mm/sec CNT100;
   1:  PR[GP1:91,1] = PR[GP1:90,1] + -66.900;
   1:  PR[GP1:91,2] = PR[GP1:90,2] + -20.922;
   1:L PR[91] R[100]mm/sec CNT100;
   1:  PR[GP1:91,1] = PR[GP1:90,1] + -66.400;
   1:  PR[GP1:91,2] = PR[GP1:90,2] + -21.574;
   1:L PR[91] R[100]mm/sec CNT100;
   1:  PR[GP1:91,1] = PR[GP1:90,1] + -58.362;
   1:  PR[GP1:91,2] = PR[GP1:90,2] + -28.891;
   1:L PR[91] R[100]mm/sec CNT100;
   1:  PR[GP1:91,1] = PR[GP1:90,1] + -57.930;
   1:  PR[GP1:91,2] = PR[GP1:90,2] + -29.152;
   1:L PR[91] R[100]mm/sec CNT100;
   1:  PR[GP1:91,1] = PR[GP1:90,1] + -57.386;
   1:  PR[GP1:91,2] = PR[GP1:90,2] + -29.354;
   1:L PR[91] R[100]mm/sec CNT100;
   1:  PR[GP1:91,1] = PR[GP1:90,1] + -47.754;
   1:  PR[GP1:91,2] = PR[GP1:90,2] + -33.527;
   1:L PR[91] R[100]mm/sec CNT100;
   1:  PR[GP1:91,1] = PR[GP1:90,1] + -47.662;
   1:  PR[GP1:91,2] = PR[GP1:90,2] + -33.542;
   1:L PR[91] R[100]mm/sec CNT100;
   1:  PR[GP1:91,1] = PR[GP1:90,1] + -43.478;
   1:  PR[GP1:91,2] = PR[GP1:90,2] + -33.857;
   1:L PR[91] R[100]mm/sec CNT100;
   1:  PR[GP1:91,1] = PR[GP1:90,1] + -36.449;
   1:  PR[GP1:91,2] = PR[GP1:90,2] + -34.434;
   1:L PR[91] R[100]mm/sec CNT100;
   1:  PR[GP1:91,1] = PR[GP1:90,1] + -35.900;
   1:  PR[GP1:91,2] = PR[GP1:90,2] + -34.345;
   1:L PR[91] R[100]mm/sec CNT100;
   1:  PR[GP1:91,1] = PR[GP1:90,1] + -25.608;
   1:  PR[GP1:91,2] = PR[GP1:90,2] + -31.756;
   1:L PR[91] R[100]mm/sec CNT100;
   1:  PR[GP1:91,1] = PR[GP1:90,1] + -24.101;
   1:  PR[GP1:91,2] = PR[GP1:90,2] + -30.986;
   1:L PR[91] R[100]mm/sec CNT100;
   1:  PR[GP1:91,1] = PR[GP1:90,1] + -16.254;
   1:  PR[GP1:91,2] = PR[GP1:90,2] + -25.890;
   1:L PR[91] R[100]mm/sec CNT100;
   1:  PR[GP1:91,1] = PR[GP1:90,1] + -14.295;
   1:  PR[GP1:91,2] = PR[GP1:90,2] + -23.925;
   1:L PR[91] R[100]mm/sec CNT100;
   1:  PR[GP1:91,1] = PR[GP1:90,1] + -9.255;
   1:  PR[GP1:91,2] = PR[GP1:90,2] + -17.454;
   1:L PR[91] R[100]mm/sec CNT100;
   1:  PR[GP1:91,1] = PR[GP1:90,1] + -7.594;
   1:  PR[GP1:91,2] = PR[GP1:90,2] + -14.137;
   1:L PR[91] R[100]mm/sec CNT100;
   1:  PR[GP1:91,1] = PR[GP1:90,1] + -5.241;
   1:  PR[GP1:91,2] = PR[GP1:90,2] + -7.207;
   1:L PR[91] R[100]mm/sec CNT100;
   1:  PR[GP1:91,1] = PR[GP1:90,1] + -4.447;
   1:  PR[GP1:91,2] = PR[GP1:90,2] + -4.972;
   1:L PR[91] R[100]mm/sec CNT100;
   1:  PR[GP1:91,1] = PR[GP1:90,1] + -2.615;
   1:  PR[GP1:91,2] = PR[GP1:90,2] + -2.947;
   1:L PR[91] R[100]mm/sec CNT100;
   1:  PR[GP1:91,1] = PR[GP1:90,1] + -2.072;
   1:  PR[GP1:91,2] = PR[GP1:90,2] + -2.615;
   1:L PR[91] R[100]mm/sec CNT100;
   1:  PR[GP1:91,1] = PR[GP1:90,1] + -1.823;
   1:  PR[GP1:91,2] = PR[GP1:90,2] + -2.319;
   1:L PR[91] R[100]mm/sec CNT100;
   1:  PR[GP1:91,1] = PR[GP1:90,1] + 2.336;
   1:  PR[GP1:91,2] = PR[GP1:90,2] + -2.639;
   1:L PR[91] R[100]mm/sec CNT100;
   1:  PR[GP1:91,1] = PR[GP1:90,1] + 2.539;
   1:  PR[GP1:91,2] = PR[GP1:90,2] + -2.803;
   1:L PR[91] R[100]mm/sec CNT100;
   1:  PR[GP1:91,1] = PR[GP1:90,1] + 2.900;
   1:  PR[GP1:91,2] = PR[GP1:90,2] + -2.799;
   1:L PR[91] R[100]mm/sec CNT100;
   1:  PR[GP1:91,1] = PR[GP1:90,1] + 4.764;
   1:  PR[GP1:91,2] = PR[GP1:90,2] + -6.346;
   1:L PR[91] R[100]mm/sec CNT100;
   1:  PR[GP1:91,1] = PR[GP1:90,1] + 5.416;
   1:  PR[GP1:91,2] = PR[GP1:90,2] + -7.099;
   1:L PR[91] R[100]mm/sec CNT100;
   1:  PR[GP1:91,1] = PR[GP1:90,1] + 7.804;
   1:  PR[GP1:91,2] = PR[GP1:90,2] + -14.132;
   1:L PR[91] R[100]mm/sec CNT100;
   1:  PR[GP1:91,1] = PR[GP1:90,1] + 9.464;
   1:  PR[GP1:91,2] = PR[GP1:90,2] + -17.444;
   1:L PR[91] R[100]mm/sec CNT100;
   1:  PR[GP1:91,1] = PR[GP1:90,1] + 14.503;
   1:  PR[GP1:91,2] = PR[GP1:90,2] + -23.917;
   1:L PR[91] R[100]mm/sec CNT100;
   1:  PR[GP1:91,1] = PR[GP1:90,1] + 16.463;
   1:  PR[GP1:91,2] = PR[GP1:90,2] + -25.888;
   1:L PR[91] R[100]mm/sec CNT100;
   1:  PR[GP1:91,1] = PR[GP1:90,1] + 24.310;
   1:  PR[GP1:91,2] = PR[GP1:90,2] + -30.983;
   1:L PR[91] R[100]mm/sec CNT100;
   1:  PR[GP1:91,1] = PR[GP1:90,1] + 25.817;
   1:  PR[GP1:91,2] = PR[GP1:90,2] + -31.754;
   1:L PR[91] R[100]mm/sec CNT100;
   1:  PR[GP1:91,1] = PR[GP1:90,1] + 36.110;
   1:  PR[GP1:91,2] = PR[GP1:90,2] + -34.344;
   1:L PR[91] R[100]mm/sec CNT100;
   1:  PR[GP1:91,1] = PR[GP1:90,1] + 36.660;
   1:  PR[GP1:91,2] = PR[GP1:90,2] + -34.434;
   1:L PR[91] R[100]mm/sec CNT100;
   1:  PR[GP1:91,1] = PR[GP1:90,1] + 43.691;
   1:  PR[GP1:91,2] = PR[GP1:90,2] + -33.857;
   1:L PR[91] R[100]mm/sec CNT100;
   1:  PR[GP1:91,1] = PR[GP1:90,1] + 47.873;
   1:  PR[GP1:91,2] = PR[GP1:90,2] + -33.543;
   1:L PR[91] R[100]mm/sec CNT100;
   1:  PR[GP1:91,1] = PR[GP1:90,1] + 47.981;
   1:  PR[GP1:91,2] = PR[GP1:90,2] + -33.524;
   1:L PR[91] R[100]mm/sec CNT100;
   1:  PR[GP1:91,1] = PR[GP1:90,1] + 48.096;
   1:  PR[GP1:91,2] = PR[GP1:90,2] + -33.482;
   1:L PR[91] R[100]mm/sec CNT100;
   1:  PR[GP1:91,1] = PR[GP1:90,1] + 58.129;
   1:  PR[GP1:91,2] = PR[GP1:90,2] + -29.161;
   1:L PR[91] R[100]mm/sec CNT100;
   1:  PR[GP1:91,1] = PR[GP1:90,1] + 58.574;
   1:  PR[GP1:91,2] = PR[GP1:90,2] + -28.893;
   1:L PR[91] R[100]mm/sec CNT100;
   1:  PR[GP1:91,1] = PR[GP1:90,1] + 66.613;
   1:  PR[GP1:91,2] = PR[GP1:90,2] + -21.573;
   1:L PR[91] R[100]mm/sec CNT100;
   1:  PR[GP1:91,1] = PR[GP1:90,1] + 67.107;
   1:  PR[GP1:91,2] = PR[GP1:90,2] + -20.928;
   1:L PR[91] R[100]mm/sec CNT100;
   1:  PR[GP1:91,1] = PR[GP1:90,1] + 67.502;
   1:  PR[GP1:91,2] = PR[GP1:90,2] + -20.146;
   1:L PR[91] R[100]mm/sec CNT100;
   1:  PR[GP1:91,1] = PR[GP1:90,1] + 72.217;
   1:  PR[GP1:91,2] = PR[GP1:90,2] + -11.496;
   1:L PR[91] R[100]mm/sec CNT100;
   1:  PR[GP1:91,1] = PR[GP1:90,1] + 72.489;
   1:  PR[GP1:91,2] = PR[GP1:90,2] + -10.555;
   1:L PR[91] R[100]mm/sec CNT100;
   1:  PR[GP1:91,1] = PR[GP1:90,1] + 72.588;
   1:  PR[GP1:91,2] = PR[GP1:90,2] + -9.492;
   1:L PR[91] R[100]mm/sec CNT100;
   1:  PR[GP1:91,1] = PR[GP1:90,1] + 74.163;
   1:  PR[GP1:91,2] = PR[GP1:90,2] + -0.050;
   1:L PR[91] R[100]mm/sec CNT100;
   1:  PR[GP1:91,1] = PR[GP1:90,1] + 74.051;
   1:  PR[GP1:91,2] = PR[GP1:90,2] + 1.141;
   1:L PR[91] R[100]mm/sec CNT100;
   1:  PR[GP1:91,1] = PR[GP1:90,1] + 72.495;
   1:  PR[GP1:91,2] = PR[GP1:90,2] + 10.389;
   1:L PR[91] R[100]mm/sec CNT100;
   1:  PR[GP1:91,1] = PR[GP1:90,1] + 72.215;
   1:  PR[GP1:91,2] = PR[GP1:90,2] + 11.361;
   1:L PR[91] R[100]mm/sec CNT100;
   1:  PR[GP1:91,1] = PR[GP1:90,1] + 71.748;
   1:  PR[GP1:91,2] = PR[GP1:90,2] + 12.286;
   1:L PR[91] R[100]mm/sec CNT100;
   1:  PR[GP1:91,1] = PR[GP1:90,1] + 67.113;
   1:  PR[GP1:91,2] = PR[GP1:90,2] + 20.776;
   1:L PR[91] R[100]mm/sec CNT100;
   1:  PR[GP1:91,1] = PR[GP1:90,1] + 66.613;
   1:  PR[GP1:91,2] = PR[GP1:90,2] + 21.429;
   1:L PR[91] R[100]mm/sec CNT100;
   1:  PR[GP1:91,1] = PR[GP1:90,1] + 58.574;
   1:  PR[GP1:91,2] = PR[GP1:90,2] + 28.749;
   1:L PR[91] R[100]mm/sec CNT100;
   1:  PR[GP1:91,1] = PR[GP1:90,1] + 58.142;
   1:  PR[GP1:91,2] = PR[GP1:90,2] + 29.009;
   1:L PR[91] R[100]mm/sec CNT100;
   1:  PR[GP1:91,1] = PR[GP1:90,1] + 57.599;
   1:  PR[GP1:91,2] = PR[GP1:90,2] + 29.211;
   1:L PR[91] R[100]mm/sec CNT100;
   1:  PR[GP1:91,1] = PR[GP1:90,1] + 47.965;
   1:  PR[GP1:91,2] = PR[GP1:90,2] + 33.383;
   1:L PR[91] R[100]mm/sec CNT100;
   1:  PR[GP1:91,1] = PR[GP1:90,1] + 47.873;
   1:  PR[GP1:91,2] = PR[GP1:90,2] + 33.399;
   1:L PR[91] R[100]mm/sec CNT100;
   1:  PR[GP1:91,1] = PR[GP1:90,1] + 43.691;
   1:  PR[GP1:91,2] = PR[GP1:90,2] + 33.713;
   1:L PR[91] R[100]mm/sec CNT100;
   1:  PR[GP1:91,1] = PR[GP1:90,1] + 36.660;
   1:  PR[GP1:91,2] = PR[GP1:90,2] + 34.290;
   1:L PR[91] R[100]mm/sec CNT100;
   1:  PR[GP1:91,1] = PR[GP1:90,1] + 36.110;
   1:  PR[GP1:91,2] = PR[GP1:90,2] + 34.200;
   1:L PR[91] R[100]mm/sec CNT100;
   1:  PR[GP1:91,1] = PR[GP1:90,1] + 25.817;
   1:  PR[GP1:91,2] = PR[GP1:90,2] + 31.610;
   1:L PR[91] R[100]mm/sec CNT100;
   1:  PR[GP1:91,1] = PR[GP1:90,1] + 24.310;
   1:  PR[GP1:91,2] = PR[GP1:90,2] + 30.839;
   1:L PR[91] R[100]mm/sec CNT100;
   1:  PR[GP1:91,1] = PR[GP1:90,1] + 16.463;
   1:  PR[GP1:91,2] = PR[GP1:90,2] + 25.744;
   1:L PR[91] R[100]mm/sec CNT100;
   1:  PR[GP1:91,1] = PR[GP1:90,1] + 14.503;
   1:  PR[GP1:91,2] = PR[GP1:90,2] + 23.773;
   1:L PR[91] R[100]mm/sec CNT100;
   1:  PR[GP1:91,1] = PR[GP1:90,1] + 9.464;
   1:  PR[GP1:91,2] = PR[GP1:90,2] + 17.300;
   1:L PR[91] R[100]mm/sec CNT100;
   1:  PR[GP1:91,1] = PR[GP1:90,1] + 7.801;
   1:  PR[GP1:91,2] = PR[GP1:90,2] + 13.980;
   1:L PR[91] R[100]mm/sec CNT100;
   1:  PR[GP1:91,1] = PR[GP1:90,1] + 5.452;
   1:  PR[GP1:91,2] = PR[GP1:90,2] + 7.062;
   1:L PR[91] R[100]mm/sec CNT100;
   1:  PR[GP1:91,1] = PR[GP1:90,1] + 4.662;
   1:  PR[GP1:91,2] = PR[GP1:90,2] + 4.837;
   1:L PR[91] R[100]mm/sec CNT100;
   1:  PR[GP1:91,1] = PR[GP1:90,1] + 4.210;
   1:  PR[GP1:91,2] = PR[GP1:90,2] + 4.289;
   1:L PR[91] R[100]mm/sec CNT100;
   1:  PR[GP1:91,1] = PR[GP1:90,1] + 2.656;
   1:  PR[GP1:91,2] = PR[GP1:90,2] + 2.599;
   1:L PR[91] R[100]mm/sec CNT100;
   1:  PR[GP1:91,1] = PR[GP1:90,1] + 1.924;
   1:  PR[GP1:91,2] = PR[GP1:90,2] + 2.194;
   1:L PR[91] R[100]mm/sec CNT100;
   1:  PR[GP1:91,1] = PR[GP1:90,1] + 1.623;
   1:  PR[GP1:91,2] = PR[GP1:90,2] + 2.197;
   1:L PR[91] R[100]mm/sec CNT100;
   1:  ! -- Layer/Ebene 30 -- !;
   1:  PR[91] = PR[90];
   1:  PR[GP1:91,1] = PR[GP1:90,1] + -2.257;
   1:  PR[GP1:91,2] = PR[GP1:90,2] + 3.007;
   1:  PR[GP1:91,3] = PR[GP1:90,3] + 18.605;
   1:L PR[91] R[100]mm/sec CNT100;
   1:  PR[GP1:91,1] = PR[GP1:90,1] + -2.703;
   1:  PR[GP1:91,2] = PR[GP1:90,2] + 3.320;
   1:L PR[91] R[100]mm/sec CNT100;
   1:  PR[GP1:91,1] = PR[GP1:90,1] + -3.154;
   1:  PR[GP1:91,2] = PR[GP1:90,2] + 3.872;
   1:L PR[91] R[100]mm/sec CNT100;
   1:  PR[GP1:91,1] = PR[GP1:90,1] + -5.200;
   1:  PR[GP1:91,2] = PR[GP1:90,2] + 7.452;
   1:L PR[91] R[100]mm/sec CNT100;
   1:  PR[GP1:91,1] = PR[GP1:90,1] + -7.234;
   1:  PR[GP1:91,2] = PR[GP1:90,2] + 13.442;
   1:L PR[91] R[100]mm/sec CNT100;
   1:  PR[GP1:91,1] = PR[GP1:90,1] + -9.334;
   1:  PR[GP1:91,2] = PR[GP1:90,2] + 17.642;
   1:L PR[91] R[100]mm/sec CNT100;
   1:  PR[GP1:91,1] = PR[GP1:90,1] + -13.772;
   1:  PR[GP1:91,2] = PR[GP1:90,2] + 23.339;
   1:L PR[91] R[100]mm/sec CNT100;
   1:  PR[GP1:91,1] = PR[GP1:90,1] + -16.382;
   1:  PR[GP1:91,2] = PR[GP1:90,2] + 25.957;
   1:L PR[91] R[100]mm/sec CNT100;
   1:  PR[GP1:91,1] = PR[GP1:90,1] + -23.451;
   1:  PR[GP1:91,2] = PR[GP1:90,2] + 30.547;
   1:L PR[91] R[100]mm/sec CNT100;
   1:  PR[GP1:91,1] = PR[GP1:90,1] + -25.737;
   1:  PR[GP1:91,2] = PR[GP1:90,2] + 31.716;
   1:L PR[91] R[100]mm/sec CNT100;
   1:  PR[GP1:91,1] = PR[GP1:90,1] + -35.190;
   1:  PR[GP1:91,2] = PR[GP1:90,2] + 34.094;
   1:L PR[91] R[100]mm/sec CNT100;
   1:  PR[GP1:91,1] = PR[GP1:90,1] + -36.549;
   1:  PR[GP1:91,2] = PR[GP1:90,2] + 34.314;
   1:L PR[91] R[100]mm/sec CNT100;
   1:  PR[GP1:91,1] = PR[GP1:90,1] + -47.465;
   1:  PR[GP1:91,2] = PR[GP1:90,2] + 33.419;
   1:L PR[91] R[100]mm/sec CNT100;
   1:  PR[GP1:91,1] = PR[GP1:90,1] + -47.755;
   1:  PR[GP1:91,2] = PR[GP1:90,2] + 33.375;
   1:L PR[91] R[100]mm/sec CNT100;
   1:  PR[GP1:91,1] = PR[GP1:90,1] + -58.111;
   1:  PR[GP1:91,2] = PR[GP1:90,2] + 28.896;
   1:L PR[91] R[100]mm/sec CNT100;
   1:  PR[GP1:91,1] = PR[GP1:90,1] + -58.241;
   1:  PR[GP1:91,2] = PR[GP1:90,2] + 28.818;
   1:L PR[91] R[100]mm/sec CNT100;
   1:  PR[GP1:91,1] = PR[GP1:90,1] + -58.381;
   1:  PR[GP1:91,2] = PR[GP1:90,2] + 28.692;
   1:L PR[91] R[100]mm/sec CNT100;
   1:  PR[GP1:91,1] = PR[GP1:90,1] + -66.481;
   1:  PR[GP1:91,2] = PR[GP1:90,2] + 21.312;
   1:L PR[91] R[100]mm/sec CNT100;
   1:  PR[GP1:91,1] = PR[GP1:90,1] + -66.760;
   1:  PR[GP1:91,2] = PR[GP1:90,2] + 20.947;
   1:L PR[91] R[100]mm/sec CNT100;
   1:  PR[GP1:91,1] = PR[GP1:90,1] + -66.996;
   1:  PR[GP1:91,2] = PR[GP1:90,2] + 20.481;
   1:L PR[91] R[100]mm/sec CNT100;
   1:  PR[GP1:91,1] = PR[GP1:90,1] + -72.010;
   1:  PR[GP1:91,2] = PR[GP1:90,2] + 11.277;
   1:L PR[91] R[100]mm/sec CNT100;
   1:  PR[GP1:91,1] = PR[GP1:90,1] + -72.186;
   1:  PR[GP1:91,2] = PR[GP1:90,2] + 10.664;
   1:L PR[91] R[100]mm/sec CNT100;
   1:  PR[GP1:91,1] = PR[GP1:90,1] + -72.254;
   1:  PR[GP1:91,2] = PR[GP1:90,2] + 9.942;
   1:L PR[91] R[100]mm/sec CNT100;
   1:  PR[GP1:91,1] = PR[GP1:90,1] + -73.928;
   1:  PR[GP1:91,2] = PR[GP1:90,2] + -0.094;
   1:L PR[91] R[100]mm/sec CNT100;
   1:  PR[GP1:91,1] = PR[GP1:90,1] + -73.847;
   1:  PR[GP1:91,2] = PR[GP1:90,2] + -0.956;
   1:L PR[91] R[100]mm/sec CNT100;
   1:  PR[GP1:91,1] = PR[GP1:90,1] + -72.192;
   1:  PR[GP1:91,2] = PR[GP1:90,2] + -10.787;
   1:L PR[91] R[100]mm/sec CNT100;
   1:  PR[GP1:91,1] = PR[GP1:90,1] + -72.007;
   1:  PR[GP1:91,2] = PR[GP1:90,2] + -11.430;
   1:L PR[91] R[100]mm/sec CNT100;
   1:  PR[GP1:91,1] = PR[GP1:90,1] + -71.695;
   1:  PR[GP1:91,2] = PR[GP1:90,2] + -12.049;
   1:L PR[91] R[100]mm/sec CNT100;
   1:  PR[GP1:91,1] = PR[GP1:90,1] + -66.766;
   1:  PR[GP1:91,2] = PR[GP1:90,2] + -21.083;
   1:L PR[91] R[100]mm/sec CNT100;
   1:  PR[GP1:91,1] = PR[GP1:90,1] + -66.481;
   1:  PR[GP1:91,2] = PR[GP1:90,2] + -21.456;
   1:L PR[91] R[100]mm/sec CNT100;
   1:  PR[GP1:91,1] = PR[GP1:90,1] + -58.238;
   1:  PR[GP1:91,2] = PR[GP1:90,2] + -28.963;
   1:L PR[91] R[100]mm/sec CNT100;
   1:  PR[GP1:91,1] = PR[GP1:90,1] + -58.125;
   1:  PR[GP1:91,2] = PR[GP1:90,2] + -29.032;
   1:L PR[91] R[100]mm/sec CNT100;
   1:  PR[GP1:91,1] = PR[GP1:90,1] + -57.930;
   1:  PR[GP1:91,2] = PR[GP1:90,2] + -29.104;
   1:L PR[91] R[100]mm/sec CNT100;
   1:  PR[GP1:91,1] = PR[GP1:90,1] + -47.755;
   1:  PR[GP1:91,2] = PR[GP1:90,2] + -33.519;
   1:L PR[91] R[100]mm/sec CNT100;
   1:  PR[GP1:91,1] = PR[GP1:90,1] + -47.465;
   1:  PR[GP1:91,2] = PR[GP1:90,2] + -33.563;
   1:L PR[91] R[100]mm/sec CNT100;
   1:  PR[GP1:91,1] = PR[GP1:90,1] + -36.549;
   1:  PR[GP1:91,2] = PR[GP1:90,2] + -34.458;
   1:L PR[91] R[100]mm/sec CNT100;
   1:  PR[GP1:91,1] = PR[GP1:90,1] + -35.190;
   1:  PR[GP1:91,2] = PR[GP1:90,2] + -34.238;
   1:L PR[91] R[100]mm/sec CNT100;
   1:  PR[GP1:91,1] = PR[GP1:90,1] + -25.737;
   1:  PR[GP1:91,2] = PR[GP1:90,2] + -31.860;
   1:L PR[91] R[100]mm/sec CNT100;
   1:  PR[GP1:91,1] = PR[GP1:90,1] + -23.451;
   1:  PR[GP1:91,2] = PR[GP1:90,2] + -30.691;
   1:L PR[91] R[100]mm/sec CNT100;
   1:  PR[GP1:91,1] = PR[GP1:90,1] + -16.382;
   1:  PR[GP1:91,2] = PR[GP1:90,2] + -26.101;
   1:L PR[91] R[100]mm/sec CNT100;
   1:  PR[GP1:91,1] = PR[GP1:90,1] + -13.772;
   1:  PR[GP1:91,2] = PR[GP1:90,2] + -23.483;
   1:L PR[91] R[100]mm/sec CNT100;
   1:  PR[GP1:91,1] = PR[GP1:90,1] + -9.334;
   1:  PR[GP1:91,2] = PR[GP1:90,2] + -17.786;
   1:L PR[91] R[100]mm/sec CNT100;
   1:  PR[GP1:91,1] = PR[GP1:90,1] + -7.237;
   1:  PR[GP1:91,2] = PR[GP1:90,2] + -13.596;
   1:L PR[91] R[100]mm/sec CNT100;
   1:  PR[GP1:91,1] = PR[GP1:90,1] + -5.217;
   1:  PR[GP1:91,2] = PR[GP1:90,2] + -7.647;
   1:L PR[91] R[100]mm/sec CNT100;
   1:  PR[GP1:91,1] = PR[GP1:90,1] + -4.481;
   1:  PR[GP1:91,2] = PR[GP1:90,2] + -5.573;
   1:L PR[91] R[100]mm/sec CNT100;
   1:  PR[GP1:91,1] = PR[GP1:90,1] + -2.786;
   1:  PR[GP1:91,2] = PR[GP1:90,2] + -3.699;
   1:L PR[91] R[100]mm/sec CNT100;
   1:  PR[GP1:91,1] = PR[GP1:90,1] + -2.287;
   1:  PR[GP1:91,2] = PR[GP1:90,2] + -3.394;
   1:L PR[91] R[100]mm/sec CNT100;
   1:  PR[GP1:91,1] = PR[GP1:90,1] + -1.833;
   1:  PR[GP1:91,2] = PR[GP1:90,2] + -2.852;
   1:L PR[91] R[100]mm/sec CNT100;
   1:  PR[GP1:91,1] = PR[GP1:90,1] + 2.089;
   1:  PR[GP1:91,2] = PR[GP1:90,2] + -3.153;
   1:L PR[91] R[100]mm/sec CNT100;
   1:  PR[GP1:91,1] = PR[GP1:90,1] + 2.277;
   1:  PR[GP1:91,2] = PR[GP1:90,2] + -3.306;
   1:L PR[91] R[100]mm/sec CNT100;
   1:  PR[GP1:91,1] = PR[GP1:90,1] + 2.855;
   1:  PR[GP1:91,2] = PR[GP1:90,2] + -3.300;
   1:L PR[91] R[100]mm/sec CNT100;
   1:  PR[GP1:91,1] = PR[GP1:90,1] + 4.608;
   1:  PR[GP1:91,2] = PR[GP1:90,2] + -6.635;
   1:L PR[91] R[100]mm/sec CNT100;
   1:  PR[GP1:91,1] = PR[GP1:90,1] + 5.391;
   1:  PR[GP1:91,2] = PR[GP1:90,2] + -7.539;
   1:L PR[91] R[100]mm/sec CNT100;
   1:  PR[GP1:91,1] = PR[GP1:90,1] + 7.446;
   1:  PR[GP1:91,2] = PR[GP1:90,2] + -13.591;
   1:L PR[91] R[100]mm/sec CNT100;
   1:  PR[GP1:91,1] = PR[GP1:90,1] + 9.542;
   1:  PR[GP1:91,2] = PR[GP1:90,2] + -17.774;
   1:L PR[91] R[100]mm/sec CNT100;
   1:  PR[GP1:91,1] = PR[GP1:90,1] + 13.980;
   1:  PR[GP1:91,2] = PR[GP1:90,2] + -23.474;
   1:L PR[91] R[100]mm/sec CNT100;
   1:  PR[GP1:91,1] = PR[GP1:90,1] + 16.590;
   1:  PR[GP1:91,2] = PR[GP1:90,2] + -26.098;
   1:L PR[91] R[100]mm/sec CNT100;
   1:  PR[GP1:91,1] = PR[GP1:90,1] + 23.659;
   1:  PR[GP1:91,2] = PR[GP1:90,2] + -30.689;
   1:L PR[91] R[100]mm/sec CNT100;
   1:  PR[GP1:91,1] = PR[GP1:90,1] + 25.946;
   1:  PR[GP1:91,2] = PR[GP1:90,2] + -31.858;
   1:L PR[91] R[100]mm/sec CNT100;
   1:  PR[GP1:91,1] = PR[GP1:90,1] + 35.399;
   1:  PR[GP1:91,2] = PR[GP1:90,2] + -34.237;
   1:L PR[91] R[100]mm/sec CNT100;
   1:  PR[GP1:91,1] = PR[GP1:90,1] + 36.759;
   1:  PR[GP1:91,2] = PR[GP1:90,2] + -34.458;
   1:L PR[91] R[100]mm/sec CNT100;
   1:  PR[GP1:91,1] = PR[GP1:90,1] + 47.676;
   1:  PR[GP1:91,2] = PR[GP1:90,2] + -33.563;
   1:L PR[91] R[100]mm/sec CNT100;
   1:  PR[GP1:91,1] = PR[GP1:90,1] + 47.967;
   1:  PR[GP1:91,2] = PR[GP1:90,2] + -33.519;
   1:L PR[91] R[100]mm/sec CNT100;
   1:  PR[GP1:91,1] = PR[GP1:90,1] + 58.323;
   1:  PR[GP1:91,2] = PR[GP1:90,2] + -29.042;
   1:L PR[91] R[100]mm/sec CNT100;
   1:  PR[GP1:91,1] = PR[GP1:90,1] + 58.450;
   1:  PR[GP1:91,2] = PR[GP1:90,2] + -28.965;
   1:L PR[91] R[100]mm/sec CNT100;
   1:  PR[GP1:91,1] = PR[GP1:90,1] + 66.694;
   1:  PR[GP1:91,2] = PR[GP1:90,2] + -21.454;
   1:L PR[91] R[100]mm/sec CNT100;
   1:  PR[GP1:91,1] = PR[GP1:90,1] + 66.973;
   1:  PR[GP1:91,2] = PR[GP1:90,2] + -21.089;
   1:L PR[91] R[100]mm/sec CNT100;
   1:  PR[GP1:91,1] = PR[GP1:90,1] + 67.209;
   1:  PR[GP1:91,2] = PR[GP1:90,2] + -20.623;
   1:L PR[91] R[100]mm/sec CNT100;
   1:  PR[GP1:91,1] = PR[GP1:90,1] + 72.223;
   1:  PR[GP1:91,2] = PR[GP1:90,2] + -11.425;
   1:L PR[91] R[100]mm/sec CNT100;
   1:  PR[GP1:91,1] = PR[GP1:90,1] + 72.399;
   1:  PR[GP1:91,2] = PR[GP1:90,2] + -10.812;
   1:L PR[91] R[100]mm/sec CNT100;
   1:  PR[GP1:91,1] = PR[GP1:90,1] + 72.467;
   1:  PR[GP1:91,2] = PR[GP1:90,2] + -10.090;
   1:L PR[91] R[100]mm/sec CNT100;
   1:  PR[GP1:91,1] = PR[GP1:90,1] + 74.141;
   1:  PR[GP1:91,2] = PR[GP1:90,2] + -0.050;
   1:L PR[91] R[100]mm/sec CNT100;
   1:  PR[GP1:91,1] = PR[GP1:90,1] + 74.060;
   1:  PR[GP1:91,2] = PR[GP1:90,2] + 0.813;
   1:L PR[91] R[100]mm/sec CNT100;
   1:  PR[GP1:91,1] = PR[GP1:90,1] + 72.406;
   1:  PR[GP1:91,2] = PR[GP1:90,2] + 10.647;
   1:L PR[91] R[100]mm/sec CNT100;
   1:  PR[GP1:91,1] = PR[GP1:90,1] + 72.220;
   1:  PR[GP1:91,2] = PR[GP1:90,2] + 11.290;
   1:L PR[91] R[100]mm/sec CNT100;
   1:  PR[GP1:91,1] = PR[GP1:90,1] + 71.908;
   1:  PR[GP1:91,2] = PR[GP1:90,2] + 11.909;
   1:L PR[91] R[100]mm/sec CNT100;
   1:  PR[GP1:91,1] = PR[GP1:90,1] + 66.979;
   1:  PR[GP1:91,2] = PR[GP1:90,2] + 20.938;
   1:L PR[91] R[100]mm/sec CNT100;
   1:  PR[GP1:91,1] = PR[GP1:90,1] + 66.694;
   1:  PR[GP1:91,2] = PR[GP1:90,2] + 21.310;
   1:L PR[91] R[100]mm/sec CNT100;
   1:  PR[GP1:91,1] = PR[GP1:90,1] + 58.450;
   1:  PR[GP1:91,2] = PR[GP1:90,2] + 28.821;
   1:L PR[91] R[100]mm/sec CNT100;
   1:  PR[GP1:91,1] = PR[GP1:90,1] + 58.337;
   1:  PR[GP1:91,2] = PR[GP1:90,2] + 28.889;
   1:L PR[91] R[100]mm/sec CNT100;
   1:  PR[GP1:91,1] = PR[GP1:90,1] + 58.143;
   1:  PR[GP1:91,2] = PR[GP1:90,2] + 28.962;
   1:L PR[91] R[100]mm/sec CNT100;
   1:  PR[GP1:91,1] = PR[GP1:90,1] + 47.967;
   1:  PR[GP1:91,2] = PR[GP1:90,2] + 33.375;
   1:L PR[91] R[100]mm/sec CNT100;
   1:  PR[GP1:91,1] = PR[GP1:90,1] + 47.676;
   1:  PR[GP1:91,2] = PR[GP1:90,2] + 33.419;
   1:L PR[91] R[100]mm/sec CNT100;
   1:  PR[GP1:91,1] = PR[GP1:90,1] + 36.759;
   1:  PR[GP1:91,2] = PR[GP1:90,2] + 34.314;
   1:L PR[91] R[100]mm/sec CNT100;
   1:  PR[GP1:91,1] = PR[GP1:90,1] + 35.399;
   1:  PR[GP1:91,2] = PR[GP1:90,2] + 34.093;
   1:L PR[91] R[100]mm/sec CNT100;
   1:  PR[GP1:91,1] = PR[GP1:90,1] + 25.946;
   1:  PR[GP1:91,2] = PR[GP1:90,2] + 31.714;
   1:L PR[91] R[100]mm/sec CNT100;
   1:  PR[GP1:91,1] = PR[GP1:90,1] + 23.659;
   1:  PR[GP1:91,2] = PR[GP1:90,2] + 30.545;
   1:L PR[91] R[100]mm/sec CNT100;
   1:  PR[GP1:91,1] = PR[GP1:90,1] + 16.590;
   1:  PR[GP1:91,2] = PR[GP1:90,2] + 25.954;
   1:L PR[91] R[100]mm/sec CNT100;
   1:  PR[GP1:91,1] = PR[GP1:90,1] + 13.980;
   1:  PR[GP1:91,2] = PR[GP1:90,2] + 23.329;
   1:L PR[91] R[100]mm/sec CNT100;
   1:  PR[GP1:91,1] = PR[GP1:90,1] + 9.542;
   1:  PR[GP1:91,2] = PR[GP1:90,2] + 17.630;
   1:L PR[91] R[100]mm/sec CNT100;
   1:  PR[GP1:91,1] = PR[GP1:90,1] + 7.443;
   1:  PR[GP1:91,2] = PR[GP1:90,2] + 13.437;
   1:L PR[91] R[100]mm/sec CNT100;
   1:  PR[GP1:91,1] = PR[GP1:90,1] + 5.427;
   1:  PR[GP1:91,2] = PR[GP1:90,2] + 7.502;
   1:L PR[91] R[100]mm/sec CNT100;
   1:  PR[GP1:91,1] = PR[GP1:90,1] + 4.695;
   1:  PR[GP1:91,2] = PR[GP1:90,2] + 5.435;
   1:L PR[91] R[100]mm/sec CNT100;
   1:  PR[GP1:91,1] = PR[GP1:90,1] + 4.087;
   1:  PR[GP1:91,2] = PR[GP1:90,2] + 4.698;
   1:L PR[91] R[100]mm/sec CNT100;
   1:  PR[GP1:91,1] = PR[GP1:90,1] + 2.628;
   1:  PR[GP1:91,2] = PR[GP1:90,2] + 3.111;
   1:L PR[91] R[100]mm/sec CNT100;
   1:  PR[GP1:91,1] = PR[GP1:90,1] + 1.929;
   1:  PR[GP1:91,2] = PR[GP1:90,2] + 2.724;
   1:L PR[91] R[100]mm/sec CNT100;
   1:  PR[GP1:91,1] = PR[GP1:90,1] + 1.406;
   1:  PR[GP1:91,2] = PR[GP1:90,2] + 2.730;
   1:L PR[91] R[100]mm/sec CNT100;
   1:  ! -- Layer/Ebene 31 -- !;
   1:  PR[91] = PR[90];
   1:  PR[GP1:91,1] = PR[GP1:90,1] + -2.234;
   1:  PR[GP1:91,2] = PR[GP1:90,2] + 3.522;
   1:  PR[GP1:91,3] = PR[GP1:90,3] + 19.215;
   1:L PR[91] R[100]mm/sec CNT100;
   1:  PR[GP1:91,1] = PR[GP1:90,1] + -2.663;
   1:  PR[GP1:91,2] = PR[GP1:90,2] + 3.823;
   1:L PR[91] R[100]mm/sec CNT100;
   1:  PR[GP1:91,1] = PR[GP1:90,1] + -3.300;
   1:  PR[GP1:91,2] = PR[GP1:90,2] + 4.603;
   1:L PR[91] R[100]mm/sec CNT100;
   1:  PR[GP1:91,1] = PR[GP1:90,1] + -5.176;
   1:  PR[GP1:91,2] = PR[GP1:90,2] + 7.892;
   1:L PR[91] R[100]mm/sec CNT100;
   1:  PR[GP1:91,1] = PR[GP1:90,1] + -6.876;
   1:  PR[GP1:91,2] = PR[GP1:90,2] + 12.899;
   1:L PR[91] R[100]mm/sec CNT100;
   1:  PR[GP1:91,1] = PR[GP1:90,1] + -9.414;
   1:  PR[GP1:91,2] = PR[GP1:90,2] + 17.974;
   1:L PR[91] R[100]mm/sec CNT100;
   1:  PR[GP1:91,1] = PR[GP1:90,1] + -13.249;
   1:  PR[GP1:91,2] = PR[GP1:90,2] + 22.898;
   1:L PR[91] R[100]mm/sec CNT100;
   1:  PR[GP1:91,1] = PR[GP1:90,1] + -16.509;
   1:  PR[GP1:91,2] = PR[GP1:90,2] + 26.167;
   1:L PR[91] R[100]mm/sec CNT100;
   1:  PR[GP1:91,1] = PR[GP1:90,1] + -22.801;
   1:  PR[GP1:91,2] = PR[GP1:90,2] + 30.253;
   1:L PR[91] R[100]mm/sec CNT100;
   1:  PR[GP1:91,1] = PR[GP1:90,1] + -25.866;
   1:  PR[GP1:91,2] = PR[GP1:90,2] + 31.820;
   1:L PR[91] R[100]mm/sec CNT100;
   1:  PR[GP1:91,1] = PR[GP1:90,1] + -34.480;
   1:  PR[GP1:91,2] = PR[GP1:90,2] + 33.987;
   1:L PR[91] R[100]mm/sec CNT100;
   1:  PR[GP1:91,1] = PR[GP1:90,1] + -36.648;
   1:  PR[GP1:91,2] = PR[GP1:90,2] + 34.338;
   1:L PR[91] R[100]mm/sec CNT100;
   1:  PR[GP1:91,1] = PR[GP1:90,1] + -46.767;
   1:  PR[GP1:91,2] = PR[GP1:90,2] + 33.509;
   1:L PR[91] R[100]mm/sec CNT100;
   1:  PR[GP1:91,1] = PR[GP1:90,1] + -47.810;
   1:  PR[GP1:91,2] = PR[GP1:90,2] + 33.350;
   1:L PR[91] R[100]mm/sec CNT100;
   1:  PR[GP1:91,1] = PR[GP1:90,1] + -58.054;
   1:  PR[GP1:91,2] = PR[GP1:90,2] + 28.897;
   1:L PR[91] R[100]mm/sec CNT100;
   1:  PR[GP1:91,1] = PR[GP1:90,1] + -58.176;
   1:  PR[GP1:91,2] = PR[GP1:90,2] + 28.836;
   1:L PR[91] R[100]mm/sec CNT100;
   1:  PR[GP1:91,1] = PR[GP1:90,1] + -66.562;
   1:  PR[GP1:91,2] = PR[GP1:90,2] + 21.193;
   1:L PR[91] R[100]mm/sec CNT100;
   1:  PR[GP1:91,1] = PR[GP1:90,1] + -66.632;
   1:  PR[GP1:91,2] = PR[GP1:90,2] + 21.101;
   1:L PR[91] R[100]mm/sec CNT100;
   1:  PR[GP1:91,1] = PR[GP1:90,1] + -72.015;
   1:  PR[GP1:91,2] = PR[GP1:90,2] + 11.205;
   1:L PR[91] R[100]mm/sec CNT100;
   1:  PR[GP1:91,1] = PR[GP1:90,1] + -72.097;
   1:  PR[GP1:91,2] = PR[GP1:90,2] + 10.921;
   1:L PR[91] R[100]mm/sec CNT100;
   1:  PR[GP1:91,1] = PR[GP1:90,1] + -72.133;
   1:  PR[GP1:91,2] = PR[GP1:90,2] + 10.540;
   1:L PR[91] R[100]mm/sec CNT100;
   1:  PR[GP1:91,1] = PR[GP1:90,1] + -73.907;
   1:  PR[GP1:91,2] = PR[GP1:90,2] + -0.094;
   1:L PR[91] R[100]mm/sec CNT100;
   1:  PR[GP1:91,1] = PR[GP1:90,1] + -73.857;
   1:  PR[GP1:91,2] = PR[GP1:90,2] + -0.628;
   1:L PR[91] R[100]mm/sec CNT100;
   1:  PR[GP1:91,1] = PR[GP1:90,1] + -72.103;
   1:  PR[GP1:91,2] = PR[GP1:90,2] + -11.044;
   1:L PR[91] R[100]mm/sec CNT100;
   1:  PR[GP1:91,1] = PR[GP1:90,1] + -72.013;
   1:  PR[GP1:91,2] = PR[GP1:90,2] + -11.358;
   1:L PR[91] R[100]mm/sec CNT100;
   1:  PR[GP1:91,1] = PR[GP1:90,1] + -71.854;
   1:  PR[GP1:91,2] = PR[GP1:90,2] + -11.673;
   1:L PR[91] R[100]mm/sec CNT100;
   1:  PR[GP1:91,1] = PR[GP1:90,1] + -66.632;
   1:  PR[GP1:91,2] = PR[GP1:90,2] + -21.245;
   1:L PR[91] R[100]mm/sec CNT100;
   1:  PR[GP1:91,1] = PR[GP1:90,1] + -66.562;
   1:  PR[GP1:91,2] = PR[GP1:90,2] + -21.337;
   1:L PR[91] R[100]mm/sec CNT100;
   1:  PR[GP1:91,1] = PR[GP1:90,1] + -58.176;
   1:  PR[GP1:91,2] = PR[GP1:90,2] + -28.980;
   1:L PR[91] R[100]mm/sec CNT100;
   1:  PR[GP1:91,1] = PR[GP1:90,1] + -58.054;
   1:  PR[GP1:91,2] = PR[GP1:90,2] + -29.041;
   1:L PR[91] R[100]mm/sec CNT100;
   1:  PR[GP1:91,1] = PR[GP1:90,1] + -47.810;
   1:  PR[GP1:91,2] = PR[GP1:90,2] + -33.494;
   1:L PR[91] R[100]mm/sec CNT100;
   1:  PR[GP1:91,1] = PR[GP1:90,1] + -46.767;
   1:  PR[GP1:91,2] = PR[GP1:90,2] + -33.653;
   1:L PR[91] R[100]mm/sec CNT100;
   1:  PR[GP1:91,1] = PR[GP1:90,1] + -36.648;
   1:  PR[GP1:91,2] = PR[GP1:90,2] + -34.482;
   1:L PR[91] R[100]mm/sec CNT100;
   1:  PR[GP1:91,1] = PR[GP1:90,1] + -34.480;
   1:  PR[GP1:91,2] = PR[GP1:90,2] + -34.131;
   1:L PR[91] R[100]mm/sec CNT100;
   1:  PR[GP1:91,1] = PR[GP1:90,1] + -25.866;
   1:  PR[GP1:91,2] = PR[GP1:90,2] + -31.965;
   1:L PR[91] R[100]mm/sec CNT100;
   1:  PR[GP1:91,1] = PR[GP1:90,1] + -22.801;
   1:  PR[GP1:91,2] = PR[GP1:90,2] + -30.397;
   1:L PR[91] R[100]mm/sec CNT100;
   1:  PR[GP1:91,1] = PR[GP1:90,1] + -16.509;
   1:  PR[GP1:91,2] = PR[GP1:90,2] + -26.311;
   1:L PR[91] R[100]mm/sec CNT100;
   1:  PR[GP1:91,1] = PR[GP1:90,1] + -13.249;
   1:  PR[GP1:91,2] = PR[GP1:90,2] + -23.042;
   1:L PR[91] R[100]mm/sec CNT100;
   1:  PR[GP1:91,1] = PR[GP1:90,1] + -9.414;
   1:  PR[GP1:91,2] = PR[GP1:90,2] + -18.118;
   1:L PR[91] R[100]mm/sec CNT100;
   1:  PR[GP1:91,1] = PR[GP1:90,1] + -6.879;
   1:  PR[GP1:91,2] = PR[GP1:90,2] + -13.055;
   1:L PR[91] R[100]mm/sec CNT100;
   1:  PR[GP1:91,1] = PR[GP1:90,1] + -5.193;
   1:  PR[GP1:91,2] = PR[GP1:90,2] + -8.087;
   1:L PR[91] R[100]mm/sec CNT100;
   1:  PR[GP1:91,1] = PR[GP1:90,1] + -4.515;
   1:  PR[GP1:91,2] = PR[GP1:90,2] + -6.173;
   1:L PR[91] R[100]mm/sec CNT100;
   1:  PR[GP1:91,1] = PR[GP1:90,1] + -2.957;
   1:  PR[GP1:91,2] = PR[GP1:90,2] + -4.451;
   1:L PR[91] R[100]mm/sec CNT100;
   1:  PR[GP1:91,1] = PR[GP1:90,1] + -2.503;
   1:  PR[GP1:91,2] = PR[GP1:90,2] + -4.173;
   1:L PR[91] R[100]mm/sec CNT100;
   1:  PR[GP1:91,1] = PR[GP1:90,1] + -1.843;
   1:  PR[GP1:91,2] = PR[GP1:90,2] + -3.385;
   1:L PR[91] R[100]mm/sec CNT100;
   1:  PR[GP1:91,1] = PR[GP1:90,1] + 1.842;
   1:  PR[GP1:91,2] = PR[GP1:90,2] + -3.668;
   1:L PR[91] R[100]mm/sec CNT100;
   1:  PR[GP1:91,1] = PR[GP1:90,1] + 2.016;
   1:  PR[GP1:91,2] = PR[GP1:90,2] + -3.809;
   1:L PR[91] R[100]mm/sec CNT100;
   1:  PR[GP1:91,1] = PR[GP1:90,1] + 2.810;
   1:  PR[GP1:91,2] = PR[GP1:90,2] + -3.801;
   1:L PR[91] R[100]mm/sec CNT100;
   1:  PR[GP1:91,1] = PR[GP1:90,1] + 4.451;
   1:  PR[GP1:91,2] = PR[GP1:90,2] + -6.924;
   1:L PR[91] R[100]mm/sec CNT100;
   1:  PR[GP1:91,1] = PR[GP1:90,1] + 5.366;
   1:  PR[GP1:91,2] = PR[GP1:90,2] + -7.978;
   1:L PR[91] R[100]mm/sec CNT100;
   1:  PR[GP1:91,1] = PR[GP1:90,1] + 7.088;
   1:  PR[GP1:91,2] = PR[GP1:90,2] + -13.050;
   1:L PR[91] R[100]mm/sec CNT100;
   1:  PR[GP1:91,1] = PR[GP1:90,1] + 9.621;
   1:  PR[GP1:91,2] = PR[GP1:90,2] + -18.104;
   1:L PR[91] R[100]mm/sec CNT100;
   1:  PR[GP1:91,1] = PR[GP1:90,1] + 13.456;
   1:  PR[GP1:91,2] = PR[GP1:90,2] + -23.030;
   1:L PR[91] R[100]mm/sec CNT100;
   1:  PR[GP1:91,1] = PR[GP1:90,1] + 16.717;
   1:  PR[GP1:91,2] = PR[GP1:90,2] + -26.309;
   1:L PR[91] R[100]mm/sec CNT100;
   1:  PR[GP1:91,1] = PR[GP1:90,1] + 23.008;
   1:  PR[GP1:91,2] = PR[GP1:90,2] + -30.394;
   1:L PR[91] R[100]mm/sec CNT100;
   1:  PR[GP1:91,1] = PR[GP1:90,1] + 26.074;
   1:  PR[GP1:91,2] = PR[GP1:90,2] + -31.962;
   1:L PR[91] R[100]mm/sec CNT100;
   1:  PR[GP1:91,1] = PR[GP1:90,1] + 34.688;
   1:  PR[GP1:91,2] = PR[GP1:90,2] + -34.129;
   1:L PR[91] R[100]mm/sec CNT100;
   1:  PR[GP1:91,1] = PR[GP1:90,1] + 36.858;
   1:  PR[GP1:91,2] = PR[GP1:90,2] + -34.482;
   1:L PR[91] R[100]mm/sec CNT100;
   1:  PR[GP1:91,1] = PR[GP1:90,1] + 46.977;
   1:  PR[GP1:91,2] = PR[GP1:90,2] + -33.653;
   1:L PR[91] R[100]mm/sec CNT100;
   1:  PR[GP1:91,1] = PR[GP1:90,1] + 48.021;
   1:  PR[GP1:91,2] = PR[GP1:90,2] + -33.495;
   1:L PR[91] R[100]mm/sec CNT100;
   1:  PR[GP1:91,1] = PR[GP1:90,1] + 58.266;
   1:  PR[GP1:91,2] = PR[GP1:90,2] + -29.043;
   1:L PR[91] R[100]mm/sec CNT100;
   1:  PR[GP1:91,1] = PR[GP1:90,1] + 58.389;
   1:  PR[GP1:91,2] = PR[GP1:90,2] + -28.982;
   1:L PR[91] R[100]mm/sec CNT100;
   1:  PR[GP1:91,1] = PR[GP1:90,1] + 66.775;
   1:  PR[GP1:91,2] = PR[GP1:90,2] + -21.335;
   1:L PR[91] R[100]mm/sec CNT100;
   1:  PR[GP1:91,1] = PR[GP1:90,1] + 66.845;
   1:  PR[GP1:91,2] = PR[GP1:90,2] + -21.243;
   1:L PR[91] R[100]mm/sec CNT100;
   1:  PR[GP1:91,1] = PR[GP1:90,1] + 72.228;
   1:  PR[GP1:91,2] = PR[GP1:90,2] + -11.354;
   1:L PR[91] R[100]mm/sec CNT100;
   1:  PR[GP1:91,1] = PR[GP1:90,1] + 72.310;
   1:  PR[GP1:91,2] = PR[GP1:90,2] + -11.070;
   1:L PR[91] R[100]mm/sec CNT100;
   1:  PR[GP1:91,1] = PR[GP1:90,1] + 72.346;
   1:  PR[GP1:91,2] = PR[GP1:90,2] + -10.688;
   1:L PR[91] R[100]mm/sec CNT100;
   1:  PR[GP1:91,1] = PR[GP1:90,1] + 74.120;
   1:  PR[GP1:91,2] = PR[GP1:90,2] + -0.050;
   1:L PR[91] R[100]mm/sec CNT100;
   1:  PR[GP1:91,1] = PR[GP1:90,1] + 74.070;
   1:  PR[GP1:91,2] = PR[GP1:90,2] + 0.484;
   1:L PR[91] R[100]mm/sec CNT100;
   1:  PR[GP1:91,1] = PR[GP1:90,1] + 72.316;
   1:  PR[GP1:91,2] = PR[GP1:90,2] + 10.904;
   1:L PR[91] R[100]mm/sec CNT100;
   1:  PR[GP1:91,1] = PR[GP1:90,1] + 72.226;
   1:  PR[GP1:91,2] = PR[GP1:90,2] + 11.219;
   1:L PR[91] R[100]mm/sec CNT100;
   1:  PR[GP1:91,1] = PR[GP1:90,1] + 72.067;
   1:  PR[GP1:91,2] = PR[GP1:90,2] + 11.533;
   1:L PR[91] R[100]mm/sec CNT100;
   1:  PR[GP1:91,1] = PR[GP1:90,1] + 66.845;
   1:  PR[GP1:91,2] = PR[GP1:90,2] + 21.099;
   1:L PR[91] R[100]mm/sec CNT100;
   1:  PR[GP1:91,1] = PR[GP1:90,1] + 66.775;
   1:  PR[GP1:91,2] = PR[GP1:90,2] + 21.191;
   1:L PR[91] R[100]mm/sec CNT100;
   1:  PR[GP1:91,1] = PR[GP1:90,1] + 58.389;
   1:  PR[GP1:91,2] = PR[GP1:90,2] + 28.838;
   1:L PR[91] R[100]mm/sec CNT100;
   1:  PR[GP1:91,1] = PR[GP1:90,1] + 58.266;
   1:  PR[GP1:91,2] = PR[GP1:90,2] + 28.899;
   1:L PR[91] R[100]mm/sec CNT100;
   1:  PR[GP1:91,1] = PR[GP1:90,1] + 48.021;
   1:  PR[GP1:91,2] = PR[GP1:90,2] + 33.351;
   1:L PR[91] R[100]mm/sec CNT100;
   1:  PR[GP1:91,1] = PR[GP1:90,1] + 46.977;
   1:  PR[GP1:91,2] = PR[GP1:90,2] + 33.509;
   1:L PR[91] R[100]mm/sec CNT100;
   1:  PR[GP1:91,1] = PR[GP1:90,1] + 36.858;
   1:  PR[GP1:91,2] = PR[GP1:90,2] + 34.338;
   1:L PR[91] R[100]mm/sec CNT100;
   1:  PR[GP1:91,1] = PR[GP1:90,1] + 34.688;
   1:  PR[GP1:91,2] = PR[GP1:90,2] + 33.985;
   1:L PR[91] R[100]mm/sec CNT100;
   1:  PR[GP1:91,1] = PR[GP1:90,1] + 26.074;
   1:  PR[GP1:91,2] = PR[GP1:90,2] + 31.818;
   1:L PR[91] R[100]mm/sec CNT100;
   1:  PR[GP1:91,1] = PR[GP1:90,1] + 23.007;
   1:  PR[GP1:91,2] = PR[GP1:90,2] + 30.250;
   1:L PR[91] R[100]mm/sec CNT100;
   1:  PR[GP1:91,1] = PR[GP1:90,1] + 16.717;
   1:  PR[GP1:91,2] = PR[GP1:90,2] + 26.165;
   1:L PR[91] R[100]mm/sec CNT100;
   1:  PR[GP1:91,1] = PR[GP1:90,1] + 13.456;
   1:  PR[GP1:91,2] = PR[GP1:90,2] + 22.886;
   1:L PR[91] R[100]mm/sec CNT100;
   1:  PR[GP1:91,1] = PR[GP1:90,1] + 9.621;
   1:  PR[GP1:91,2] = PR[GP1:90,2] + 17.960;
   1:L PR[91] R[100]mm/sec CNT100;
   1:  PR[GP1:91,1] = PR[GP1:90,1] + 7.084;
   1:  PR[GP1:91,2] = PR[GP1:90,2] + 12.894;
   1:L PR[91] R[100]mm/sec CNT100;
   1:  PR[GP1:91,1] = PR[GP1:90,1] + 5.403;
   1:  PR[GP1:91,2] = PR[GP1:90,2] + 7.942;
   1:L PR[91] R[100]mm/sec CNT100;
   1:  PR[GP1:91,1] = PR[GP1:90,1] + 4.728;
   1:  PR[GP1:91,2] = PR[GP1:90,2] + 6.033;
   1:L PR[91] R[100]mm/sec CNT100;
   1:  PR[GP1:91,1] = PR[GP1:90,1] + 3.963;
   1:  PR[GP1:91,2] = PR[GP1:90,2] + 5.107;
   1:L PR[91] R[100]mm/sec CNT100;
   1:  PR[GP1:91,1] = PR[GP1:90,1] + 2.600;
   1:  PR[GP1:91,2] = PR[GP1:90,2] + 3.624;
   1:L PR[91] R[100]mm/sec CNT100;
   1:  PR[GP1:91,1] = PR[GP1:90,1] + 1.933;
   1:  PR[GP1:91,2] = PR[GP1:90,2] + 3.255;
   1:L PR[91] R[100]mm/sec CNT100;
   1:  PR[GP1:91,1] = PR[GP1:90,1] + 1.188;
   1:  PR[GP1:91,2] = PR[GP1:90,2] + 3.263;
   1:L PR[91] R[100]mm/sec CNT100;
   1:  ! -- Layer/Ebene 32 -- !;
   1:  PR[91] = PR[90];
   1:  PR[GP1:91,1] = PR[GP1:90,1] + -2.211;
   1:  PR[GP1:91,2] = PR[GP1:90,2] + 4.037;
   1:  PR[GP1:91,3] = PR[GP1:90,3] + 19.825;
   1:L PR[91] R[100]mm/sec CNT100;
   1:  PR[GP1:91,1] = PR[GP1:90,1] + -2.623;
   1:  PR[GP1:91,2] = PR[GP1:90,2] + 4.326;
   1:L PR[91] R[100]mm/sec CNT100;
   1:  PR[GP1:91,1] = PR[GP1:90,1] + -3.446;
   1:  PR[GP1:91,2] = PR[GP1:90,2] + 5.334;
   1:L PR[91] R[100]mm/sec CNT100;
   1:  PR[GP1:91,1] = PR[GP1:90,1] + -5.152;
   1:  PR[GP1:91,2] = PR[GP1:90,2] + 8.333;
   1:L PR[91] R[100]mm/sec CNT100;
   1:  PR[GP1:91,1] = PR[GP1:90,1] + -6.518;
   1:  PR[GP1:91,2] = PR[GP1:90,2] + 12.356;
   1:L PR[91] R[100]mm/sec CNT100;
   1:  PR[GP1:91,1] = PR[GP1:90,1] + -9.493;
   1:  PR[GP1:91,2] = PR[GP1:90,2] + 18.306;
   1:L PR[91] R[100]mm/sec CNT100;
   1:  PR[GP1:91,1] = PR[GP1:90,1] + -12.726;
   1:  PR[GP1:91,2] = PR[GP1:90,2] + 22.457;
   1:L PR[91] R[100]mm/sec CNT100;
   1:  PR[GP1:91,1] = PR[GP1:90,1] + -16.637;
   1:  PR[GP1:91,2] = PR[GP1:90,2] + 26.378;
   1:L PR[91] R[100]mm/sec CNT100;
   1:  PR[GP1:91,1] = PR[GP1:90,1] + -22.150;
   1:  PR[GP1:91,2] = PR[GP1:90,2] + 29.959;
   1:L PR[91] R[100]mm/sec CNT100;
   1:  PR[GP1:91,1] = PR[GP1:90,1] + -25.995;
   1:  PR[GP1:91,2] = PR[GP1:90,2] + 31.925;
   1:L PR[91] R[100]mm/sec CNT100;
   1:  PR[GP1:91,1] = PR[GP1:90,1] + -33.770;
   1:  PR[GP1:91,2] = PR[GP1:90,2] + 33.880;
   1:L PR[91] R[100]mm/sec CNT100;
   1:  PR[GP1:91,1] = PR[GP1:90,1] + -36.748;
   1:  PR[GP1:91,2] = PR[GP1:90,2] + 34.363;
   1:L PR[91] R[100]mm/sec CNT100;
   1:  PR[GP1:91,1] = PR[GP1:90,1] + -46.068;
   1:  PR[GP1:91,2] = PR[GP1:90,2] + 33.599;
   1:L PR[91] R[100]mm/sec CNT100;
   1:  PR[GP1:91,1] = PR[GP1:90,1] + -47.865;
   1:  PR[GP1:91,2] = PR[GP1:90,2] + 33.326;
   1:L PR[91] R[100]mm/sec CNT100;
   1:  PR[GP1:91,1] = PR[GP1:90,1] + -57.430;
   1:  PR[GP1:91,2] = PR[GP1:90,2] + 29.168;
   1:L PR[91] R[100]mm/sec CNT100;
   1:  PR[GP1:91,1] = PR[GP1:90,1] + -58.184;
   1:  PR[GP1:91,2] = PR[GP1:90,2] + 28.791;
   1:L PR[91] R[100]mm/sec CNT100;
   1:  PR[GP1:91,1] = PR[GP1:90,1] + -66.564;
   1:  PR[GP1:91,2] = PR[GP1:90,2] + 21.135;
   1:L PR[91] R[100]mm/sec CNT100;
   1:  PR[GP1:91,1] = PR[GP1:90,1] + -72.004;
   1:  PR[GP1:91,2] = PR[GP1:90,2] + 11.165;
   1:L PR[91] R[100]mm/sec CNT100;
   1:  PR[GP1:91,1] = PR[GP1:90,1] + -73.885;
   1:  PR[GP1:91,2] = PR[GP1:90,2] + -0.094;
   1:L PR[91] R[100]mm/sec CNT100;
   1:  PR[GP1:91,1] = PR[GP1:90,1] + -73.866;
   1:  PR[GP1:91,2] = PR[GP1:90,2] + -0.300;
   1:L PR[91] R[100]mm/sec CNT100;
   1:  PR[GP1:91,1] = PR[GP1:90,1] + -72.019;
   1:  PR[GP1:91,2] = PR[GP1:90,2] + -11.273;
   1:L PR[91] R[100]mm/sec CNT100;
   1:  PR[GP1:91,1] = PR[GP1:90,1] + -72.000;
   1:  PR[GP1:91,2] = PR[GP1:90,2] + -11.321;
   1:L PR[91] R[100]mm/sec CNT100;
   1:  PR[GP1:91,1] = PR[GP1:90,1] + -70.045;
   1:  PR[GP1:91,2] = PR[GP1:90,2] + -14.904;
   1:L PR[91] R[100]mm/sec CNT100;
   1:  PR[GP1:91,1] = PR[GP1:90,1] + -66.564;
   1:  PR[GP1:91,2] = PR[GP1:90,2] + -21.279;
   1:L PR[91] R[100]mm/sec CNT100;
   1:  PR[GP1:91,1] = PR[GP1:90,1] + -58.184;
   1:  PR[GP1:91,2] = PR[GP1:90,2] + -28.935;
   1:L PR[91] R[100]mm/sec CNT100;
   1:  PR[GP1:91,1] = PR[GP1:90,1] + -57.430;
   1:  PR[GP1:91,2] = PR[GP1:90,2] + -29.312;
   1:L PR[91] R[100]mm/sec CNT100;
   1:  PR[GP1:91,1] = PR[GP1:90,1] + -47.865;
   1:  PR[GP1:91,2] = PR[GP1:90,2] + -33.470;
   1:L PR[91] R[100]mm/sec CNT100;
   1:  PR[GP1:91,1] = PR[GP1:90,1] + -46.068;
   1:  PR[GP1:91,2] = PR[GP1:90,2] + -33.743;
   1:L PR[91] R[100]mm/sec CNT100;
   1:  PR[GP1:91,1] = PR[GP1:90,1] + -36.748;
   1:  PR[GP1:91,2] = PR[GP1:90,2] + -34.507;
   1:L PR[91] R[100]mm/sec CNT100;
   1:  PR[GP1:91,1] = PR[GP1:90,1] + -33.770;
   1:  PR[GP1:91,2] = PR[GP1:90,2] + -34.024;
   1:L PR[91] R[100]mm/sec CNT100;
   1:  PR[GP1:91,1] = PR[GP1:90,1] + -25.995;
   1:  PR[GP1:91,2] = PR[GP1:90,2] + -32.069;
   1:L PR[91] R[100]mm/sec CNT100;
   1:  PR[GP1:91,1] = PR[GP1:90,1] + -22.151;
   1:  PR[GP1:91,2] = PR[GP1:90,2] + -30.103;
   1:L PR[91] R[100]mm/sec CNT100;
   1:  PR[GP1:91,1] = PR[GP1:90,1] + -16.637;
   1:  PR[GP1:91,2] = PR[GP1:90,2] + -26.522;
   1:L PR[91] R[100]mm/sec CNT100;
   1:  PR[GP1:91,1] = PR[GP1:90,1] + -12.726;
   1:  PR[GP1:91,2] = PR[GP1:90,2] + -22.601;
   1:L PR[91] R[100]mm/sec CNT100;
   1:  PR[GP1:91,1] = PR[GP1:90,1] + -9.493;
   1:  PR[GP1:91,2] = PR[GP1:90,2] + -18.450;
   1:L PR[91] R[100]mm/sec CNT100;
   1:  PR[GP1:91,1] = PR[GP1:90,1] + -6.522;
   1:  PR[GP1:91,2] = PR[GP1:90,2] + -12.513;
   1:L PR[91] R[100]mm/sec CNT100;
   1:  PR[GP1:91,1] = PR[GP1:90,1] + -5.169;
   1:  PR[GP1:91,2] = PR[GP1:90,2] + -8.527;
   1:L PR[91] R[100]mm/sec CNT100;
   1:  PR[GP1:91,1] = PR[GP1:90,1] + -4.549;
   1:  PR[GP1:91,2] = PR[GP1:90,2] + -6.774;
   1:L PR[91] R[100]mm/sec CNT100;
   1:  PR[GP1:91,1] = PR[GP1:90,1] + -3.128;
   1:  PR[GP1:91,2] = PR[GP1:90,2] + -5.202;
   1:L PR[91] R[100]mm/sec CNT100;
   1:  PR[GP1:91,1] = PR[GP1:90,1] + -2.719;
   1:  PR[GP1:91,2] = PR[GP1:90,2] + -4.952;
   1:L PR[91] R[100]mm/sec CNT100;
   1:  PR[GP1:91,1] = PR[GP1:90,1] + -1.853;
   1:  PR[GP1:91,2] = PR[GP1:90,2] + -3.918;
   1:L PR[91] R[100]mm/sec CNT100;
   1:  PR[GP1:91,1] = PR[GP1:90,1] + 1.595;
   1:  PR[GP1:91,2] = PR[GP1:90,2] + -4.183;
   1:L PR[91] R[100]mm/sec CNT100;
   1:  PR[GP1:91,1] = PR[GP1:90,1] + 1.754;
   1:  PR[GP1:91,2] = PR[GP1:90,2] + -4.312;
   1:L PR[91] R[100]mm/sec CNT100;
   1:  PR[GP1:91,1] = PR[GP1:90,1] + 2.766;
   1:  PR[GP1:91,2] = PR[GP1:90,2] + -4.301;
   1:L PR[91] R[100]mm/sec CNT100;
   1:  PR[GP1:91,1] = PR[GP1:90,1] + 4.295;
   1:  PR[GP1:91,2] = PR[GP1:90,2] + -7.212;
   1:L PR[91] R[100]mm/sec CNT100;
   1:  PR[GP1:91,1] = PR[GP1:90,1] + 5.341;
   1:  PR[GP1:91,2] = PR[GP1:90,2] + -8.418;
   1:L PR[91] R[100]mm/sec CNT100;
   1:  PR[GP1:91,1] = PR[GP1:90,1] + 6.730;
   1:  PR[GP1:91,2] = PR[GP1:90,2] + -12.508;
   1:L PR[91] R[100]mm/sec CNT100;
   1:  PR[GP1:91,1] = PR[GP1:90,1] + 9.700;
   1:  PR[GP1:91,2] = PR[GP1:90,2] + -18.434;
   1:L PR[91] R[100]mm/sec CNT100;
   1:  PR[GP1:91,1] = PR[GP1:90,1] + 12.933;
   1:  PR[GP1:91,2] = PR[GP1:90,2] + -22.587;
   1:L PR[91] R[100]mm/sec CNT100;
   1:  PR[GP1:91,1] = PR[GP1:90,1] + 16.844;
   1:  PR[GP1:91,2] = PR[GP1:90,2] + -26.519;
   1:L PR[91] R[100]mm/sec CNT100;
   1:  PR[GP1:91,1] = PR[GP1:90,1] + 22.356;
   1:  PR[GP1:91,2] = PR[GP1:90,2] + -30.099;
   1:L PR[91] R[100]mm/sec CNT100;
   1:  PR[GP1:91,1] = PR[GP1:90,1] + 26.203;
   1:  PR[GP1:91,2] = PR[GP1:90,2] + -32.066;
   1:L PR[91] R[100]mm/sec CNT100;
   1:  PR[GP1:91,1] = PR[GP1:90,1] + 33.977;
   1:  PR[GP1:91,2] = PR[GP1:90,2] + -34.022;
   1:L PR[91] R[100]mm/sec CNT100;
   1:  PR[GP1:91,1] = PR[GP1:90,1] + 36.957;
   1:  PR[GP1:91,2] = PR[GP1:90,2] + -34.507;
   1:L PR[91] R[100]mm/sec CNT100;
   1:  PR[GP1:91,1] = PR[GP1:90,1] + 46.278;
   1:  PR[GP1:91,2] = PR[GP1:90,2] + -33.743;
   1:L PR[91] R[100]mm/sec CNT100;
   1:  PR[GP1:91,1] = PR[GP1:90,1] + 48.075;
   1:  PR[GP1:91,2] = PR[GP1:90,2] + -33.470;
   1:L PR[91] R[100]mm/sec CNT100;
   1:  PR[GP1:91,1] = PR[GP1:90,1] + 57.642;
   1:  PR[GP1:91,2] = PR[GP1:90,2] + -29.313;
   1:L PR[91] R[100]mm/sec CNT100;
   1:  PR[GP1:91,1] = PR[GP1:90,1] + 58.396;
   1:  PR[GP1:91,2] = PR[GP1:90,2] + -28.937;
   1:L PR[91] R[100]mm/sec CNT100;
   1:  PR[GP1:91,1] = PR[GP1:90,1] + 66.777;
   1:  PR[GP1:91,2] = PR[GP1:90,2] + -21.277;
   1:L PR[91] R[100]mm/sec CNT100;
   1:  PR[GP1:91,1] = PR[GP1:90,1] + 72.217;
   1:  PR[GP1:91,2] = PR[GP1:90,2] + -11.313;
   1:L PR[91] R[100]mm/sec CNT100;
   1:  PR[GP1:91,1] = PR[GP1:90,1] + 74.099;
   1:  PR[GP1:91,2] = PR[GP1:90,2] + -0.050;
   1:L PR[91] R[100]mm/sec CNT100;
   1:  PR[GP1:91,1] = PR[GP1:90,1] + 74.079;
   1:  PR[GP1:91,2] = PR[GP1:90,2] + 0.156;
   1:L PR[91] R[100]mm/sec CNT100;
   1:  PR[GP1:91,1] = PR[GP1:90,1] + 72.217;
   1:  PR[GP1:91,2] = PR[GP1:90,2] + 11.169;
   1:L PR[91] R[100]mm/sec CNT100;
   1:  PR[GP1:91,1] = PR[GP1:90,1] + 66.777;
   1:  PR[GP1:91,2] = PR[GP1:90,2] + 21.133;
   1:L PR[91] R[100]mm/sec CNT100;
   1:  PR[GP1:91,1] = PR[GP1:90,1] + 58.396;
   1:  PR[GP1:91,2] = PR[GP1:90,2] + 28.793;
   1:L PR[91] R[100]mm/sec CNT100;
   1:  PR[GP1:91,1] = PR[GP1:90,1] + 57.642;
   1:  PR[GP1:91,2] = PR[GP1:90,2] + 29.169;
   1:L PR[91] R[100]mm/sec CNT100;
   1:  PR[GP1:91,1] = PR[GP1:90,1] + 48.075;
   1:  PR[GP1:91,2] = PR[GP1:90,2] + 33.326;
   1:L PR[91] R[100]mm/sec CNT100;
   1:  PR[GP1:91,1] = PR[GP1:90,1] + 46.278;
   1:  PR[GP1:91,2] = PR[GP1:90,2] + 33.599;
   1:L PR[91] R[100]mm/sec CNT100;
   1:  PR[GP1:91,1] = PR[GP1:90,1] + 36.957;
   1:  PR[GP1:91,2] = PR[GP1:90,2] + 34.363;
   1:L PR[91] R[100]mm/sec CNT100;
   1:  PR[GP1:91,1] = PR[GP1:90,1] + 33.977;
   1:  PR[GP1:91,2] = PR[GP1:90,2] + 33.878;
   1:L PR[91] R[100]mm/sec CNT100;
   1:  PR[GP1:91,1] = PR[GP1:90,1] + 26.203;
   1:  PR[GP1:91,2] = PR[GP1:90,2] + 31.922;
   1:L PR[91] R[100]mm/sec CNT100;
   1:  PR[GP1:91,1] = PR[GP1:90,1] + 22.356;
   1:  PR[GP1:91,2] = PR[GP1:90,2] + 29.955;
   1:L PR[91] R[100]mm/sec CNT100;
   1:  PR[GP1:91,1] = PR[GP1:90,1] + 16.844;
   1:  PR[GP1:91,2] = PR[GP1:90,2] + 26.375;
   1:L PR[91] R[100]mm/sec CNT100;
   1:  PR[GP1:91,1] = PR[GP1:90,1] + 12.933;
   1:  PR[GP1:91,2] = PR[GP1:90,2] + 22.442;
   1:L PR[91] R[100]mm/sec CNT100;
   1:  PR[GP1:91,1] = PR[GP1:90,1] + 9.700;
   1:  PR[GP1:91,2] = PR[GP1:90,2] + 18.290;
   1:L PR[91] R[100]mm/sec CNT100;
   1:  PR[GP1:91,1] = PR[GP1:90,1] + 6.726;
   1:  PR[GP1:91,2] = PR[GP1:90,2] + 12.351;
   1:L PR[91] R[100]mm/sec CNT100;
   1:  PR[GP1:91,1] = PR[GP1:90,1] + 5.378;
   1:  PR[GP1:91,2] = PR[GP1:90,2] + 8.383;
   1:L PR[91] R[100]mm/sec CNT100;
   1:  PR[GP1:91,1] = PR[GP1:90,1] + 4.761;
   1:  PR[GP1:91,2] = PR[GP1:90,2] + 6.631;
   1:L PR[91] R[100]mm/sec CNT100;
   1:  PR[GP1:91,1] = PR[GP1:90,1] + 3.840;
   1:  PR[GP1:91,2] = PR[GP1:90,2] + 5.516;
   1:L PR[91] R[100]mm/sec CNT100;
   1:  PR[GP1:91,1] = PR[GP1:90,1] + 2.572;
   1:  PR[GP1:91,2] = PR[GP1:90,2] + 4.137;
   1:L PR[91] R[100]mm/sec CNT100;
   1:  PR[GP1:91,1] = PR[GP1:90,1] + 1.938;
   1:  PR[GP1:91,2] = PR[GP1:90,2] + 3.786;
   1:L PR[91] R[100]mm/sec CNT100;
   1:  PR[GP1:91,1] = PR[GP1:90,1] + 0.971;
   1:  PR[GP1:91,2] = PR[GP1:90,2] + 3.796;
   1:L PR[91] R[100]mm/sec CNT100;
   1:  ! -- Layer/Ebene 33 -- !;
   1:  PR[91] = PR[90];
   1:  PR[GP1:91,1] = PR[GP1:90,1] + -2.188;
   1:  PR[GP1:91,2] = PR[GP1:90,2] + 4.552;
   1:  PR[GP1:91,3] = PR[GP1:90,3] + 20.435;
   1:L PR[91] R[100]mm/sec CNT100;
   1:  PR[GP1:91,1] = PR[GP1:90,1] + -2.584;
   1:  PR[GP1:91,2] = PR[GP1:90,2] + 4.829;
   1:L PR[91] R[100]mm/sec CNT100;
   1:  PR[GP1:91,1] = PR[GP1:90,1] + -3.592;
   1:  PR[GP1:91,2] = PR[GP1:90,2] + 6.066;
   1:L PR[91] R[100]mm/sec CNT100;
   1:  PR[GP1:91,1] = PR[GP1:90,1] + -5.128;
   1:  PR[GP1:91,2] = PR[GP1:90,2] + 8.773;
   1:L PR[91] R[100]mm/sec CNT100;
   1:  PR[GP1:91,1] = PR[GP1:90,1] + -6.160;
   1:  PR[GP1:91,2] = PR[GP1:90,2] + 11.813;
   1:L PR[91] R[100]mm/sec CNT100;
   1:  PR[GP1:91,1] = PR[GP1:90,1] + -9.573;
   1:  PR[GP1:91,2] = PR[GP1:90,2] + 18.637;
   1:L PR[91] R[100]mm/sec CNT100;
   1:  PR[GP1:91,1] = PR[GP1:90,1] + -12.204;
   1:  PR[GP1:91,2] = PR[GP1:90,2] + 22.015;
   1:L PR[91] R[100]mm/sec CNT100;
   1:  PR[GP1:91,1] = PR[GP1:90,1] + -16.765;
   1:  PR[GP1:91,2] = PR[GP1:90,2] + 26.589;
   1:L PR[91] R[100]mm/sec CNT100;
   1:  PR[GP1:91,1] = PR[GP1:90,1] + -21.500;
   1:  PR[GP1:91,2] = PR[GP1:90,2] + 29.664;
   1:L PR[91] R[100]mm/sec CNT100;
   1:  PR[GP1:91,1] = PR[GP1:90,1] + -26.124;
   1:  PR[GP1:91,2] = PR[GP1:90,2] + 32.029;
   1:L PR[91] R[100]mm/sec CNT100;
   1:  PR[GP1:91,1] = PR[GP1:90,1] + -33.059;
   1:  PR[GP1:91,2] = PR[GP1:90,2] + 33.773;
   1:L PR[91] R[100]mm/sec CNT100;
   1:  PR[GP1:91,1] = PR[GP1:90,1] + -36.847;
   1:  PR[GP1:91,2] = PR[GP1:90,2] + 34.387;
   1:L PR[91] R[100]mm/sec CNT100;
   1:  PR[GP1:91,1] = PR[GP1:90,1] + -45.370;
   1:  PR[GP1:91,2] = PR[GP1:90,2] + 33.688;
   1:L PR[91] R[100]mm/sec CNT100;
   1:  PR[GP1:91,1] = PR[GP1:90,1] + -47.920;
   1:  PR[GP1:91,2] = PR[GP1:90,2] + 33.301;
   1:L PR[91] R[100]mm/sec CNT100;
   1:  PR[GP1:91,1] = PR[GP1:90,1] + -56.807;
   1:  PR[GP1:91,2] = PR[GP1:90,2] + 29.438;
   1:L PR[91] R[100]mm/sec CNT100;
   1:  PR[GP1:91,1] = PR[GP1:90,1] + -58.193;
   1:  PR[GP1:91,2] = PR[GP1:90,2] + 28.746;
   1:L PR[91] R[100]mm/sec CNT100;
   1:  PR[GP1:91,1] = PR[GP1:90,1] + -65.949;
   1:  PR[GP1:91,2] = PR[GP1:90,2] + 21.672;
   1:L PR[91] R[100]mm/sec CNT100;
   1:  PR[GP1:91,1] = PR[GP1:90,1] + -66.528;
   1:  PR[GP1:91,2] = PR[GP1:90,2] + 21.102;
   1:L PR[91] R[100]mm/sec CNT100;
   1:  PR[GP1:91,1] = PR[GP1:90,1] + -71.786;
   1:  PR[GP1:91,2] = PR[GP1:90,2] + 11.472;
   1:L PR[91] R[100]mm/sec CNT100;
   1:  PR[GP1:91,1] = PR[GP1:90,1] + -71.960;
   1:  PR[GP1:91,2] = PR[GP1:90,2] + 11.135;
   1:L PR[91] R[100]mm/sec CNT100;
   1:  PR[GP1:91,1] = PR[GP1:90,1] + -73.857;
   1:  PR[GP1:91,2] = PR[GP1:90,2] + -0.072;
   1:L PR[91] R[100]mm/sec CNT100;
   1:  PR[GP1:91,1] = PR[GP1:90,1] + -72.014;
   1:  PR[GP1:91,2] = PR[GP1:90,2] + -10.939;
   1:L PR[91] R[100]mm/sec CNT100;
   1:  PR[GP1:91,1] = PR[GP1:90,1] + -71.959;
   1:  PR[GP1:91,2] = PR[GP1:90,2] + -11.282;
   1:L PR[91] R[100]mm/sec CNT100;
   1:  PR[GP1:91,1] = PR[GP1:90,1] + -71.786;
   1:  PR[GP1:91,2] = PR[GP1:90,2] + -11.617;
   1:L PR[91] R[100]mm/sec CNT100;
   1:  PR[GP1:91,1] = PR[GP1:90,1] + -66.528;
   1:  PR[GP1:91,2] = PR[GP1:90,2] + -21.246;
   1:L PR[91] R[100]mm/sec CNT100;
   1:  PR[GP1:91,1] = PR[GP1:90,1] + -65.949;
   1:  PR[GP1:91,2] = PR[GP1:90,2] + -21.816;
   1:L PR[91] R[100]mm/sec CNT100;
   1:  PR[GP1:91,1] = PR[GP1:90,1] + -58.193;
   1:  PR[GP1:91,2] = PR[GP1:90,2] + -28.890;
   1:L PR[91] R[100]mm/sec CNT100;
   1:  PR[GP1:91,1] = PR[GP1:90,1] + -56.807;
   1:  PR[GP1:91,2] = PR[GP1:90,2] + -29.582;
   1:L PR[91] R[100]mm/sec CNT100;
   1:  PR[GP1:91,1] = PR[GP1:90,1] + -47.920;
   1:  PR[GP1:91,2] = PR[GP1:90,2] + -33.445;
   1:L PR[91] R[100]mm/sec CNT100;
   1:  PR[GP1:91,1] = PR[GP1:90,1] + -45.370;
   1:  PR[GP1:91,2] = PR[GP1:90,2] + -33.832;
   1:L PR[91] R[100]mm/sec CNT100;
   1:  PR[GP1:91,1] = PR[GP1:90,1] + -36.847;
   1:  PR[GP1:91,2] = PR[GP1:90,2] + -34.531;
   1:L PR[91] R[100]mm/sec CNT100;
   1:  PR[GP1:91,1] = PR[GP1:90,1] + -33.059;
   1:  PR[GP1:91,2] = PR[GP1:90,2] + -33.917;
   1:L PR[91] R[100]mm/sec CNT100;
   1:  PR[GP1:91,1] = PR[GP1:90,1] + -26.125;
   1:  PR[GP1:91,2] = PR[GP1:90,2] + -32.173;
   1:L PR[91] R[100]mm/sec CNT100;
   1:  PR[GP1:91,1] = PR[GP1:90,1] + -21.500;
   1:  PR[GP1:91,2] = PR[GP1:90,2] + -29.808;
   1:L PR[91] R[100]mm/sec CNT100;
   1:  PR[GP1:91,1] = PR[GP1:90,1] + -16.765;
   1:  PR[GP1:91,2] = PR[GP1:90,2] + -26.733;
   1:L PR[91] R[100]mm/sec CNT100;
   1:  PR[GP1:91,1] = PR[GP1:90,1] + -12.204;
   1:  PR[GP1:91,2] = PR[GP1:90,2] + -22.159;
   1:L PR[91] R[100]mm/sec CNT100;
   1:  PR[GP1:91,1] = PR[GP1:90,1] + -9.573;
   1:  PR[GP1:91,2] = PR[GP1:90,2] + -18.781;
   1:L PR[91] R[100]mm/sec CNT100;
   1:  PR[GP1:91,1] = PR[GP1:90,1] + -6.165;
   1:  PR[GP1:91,2] = PR[GP1:90,2] + -11.972;
   1:L PR[91] R[100]mm/sec CNT100;
   1:  PR[GP1:91,1] = PR[GP1:90,1] + -5.145;
   1:  PR[GP1:91,2] = PR[GP1:90,2] + -8.967;
   1:L PR[91] R[100]mm/sec CNT100;
   1:  PR[GP1:91,1] = PR[GP1:90,1] + -4.583;
   1:  PR[GP1:91,2] = PR[GP1:90,2] + -7.374;
   1:L PR[91] R[100]mm/sec CNT100;
   1:  PR[GP1:91,1] = PR[GP1:90,1] + -3.299;
   1:  PR[GP1:91,2] = PR[GP1:90,2] + -5.954;
   1:L PR[91] R[100]mm/sec CNT100;
   1:  PR[GP1:91,1] = PR[GP1:90,1] + -2.934;
   1:  PR[GP1:91,2] = PR[GP1:90,2] + -5.731;
   1:L PR[91] R[100]mm/sec CNT100;
   1:  PR[GP1:91,1] = PR[GP1:90,1] + -1.863;
   1:  PR[GP1:91,2] = PR[GP1:90,2] + -4.451;
   1:L PR[91] R[100]mm/sec CNT100;
   1:  PR[GP1:91,1] = PR[GP1:90,1] + 1.348;
   1:  PR[GP1:91,2] = PR[GP1:90,2] + -4.698;
   1:L PR[91] R[100]mm/sec CNT100;
   1:  PR[GP1:91,1] = PR[GP1:90,1] + 1.493;
   1:  PR[GP1:91,2] = PR[GP1:90,2] + -4.815;
   1:L PR[91] R[100]mm/sec CNT100;
   1:  PR[GP1:91,1] = PR[GP1:90,1] + 2.721;
   1:  PR[GP1:91,2] = PR[GP1:90,2] + -4.802;
   1:L PR[91] R[100]mm/sec CNT100;
   1:  PR[GP1:91,1] = PR[GP1:90,1] + 4.139;
   1:  PR[GP1:91,2] = PR[GP1:90,2] + -7.501;
   1:L PR[91] R[100]mm/sec CNT100;
   1:  PR[GP1:91,1] = PR[GP1:90,1] + 5.317;
   1:  PR[GP1:91,2] = PR[GP1:90,2] + -8.858;
   1:L PR[91] R[100]mm/sec CNT100;
   1:  PR[GP1:91,1] = PR[GP1:90,1] + 6.372;
   1:  PR[GP1:91,2] = PR[GP1:90,2] + -11.967;
   1:L PR[91] R[100]mm/sec CNT100;
   1:  PR[GP1:91,1] = PR[GP1:90,1] + 9.779;
   1:  PR[GP1:91,2] = PR[GP1:90,2] + -18.764;
   1:L PR[91] R[100]mm/sec CNT100;
   1:  PR[GP1:91,1] = PR[GP1:90,1] + 12.409;
   1:  PR[GP1:91,2] = PR[GP1:90,2] + -22.143;
   1:L PR[91] R[100]mm/sec CNT100;
   1:  PR[GP1:91,1] = PR[GP1:90,1] + 16.971;
   1:  PR[GP1:91,2] = PR[GP1:90,2] + -26.730;
   1:L PR[91] R[100]mm/sec CNT100;
   1:  PR[GP1:91,1] = PR[GP1:90,1] + 21.705;
   1:  PR[GP1:91,2] = PR[GP1:90,2] + -29.804;
   1:L PR[91] R[100]mm/sec CNT100;
   1:  PR[GP1:91,1] = PR[GP1:90,1] + 26.331;
   1:  PR[GP1:91,2] = PR[GP1:90,2] + -32.170;
   1:L PR[91] R[100]mm/sec CNT100;
   1:  PR[GP1:91,1] = PR[GP1:90,1] + 33.266;
   1:  PR[GP1:91,2] = PR[GP1:90,2] + -33.915;
   1:L PR[91] R[100]mm/sec CNT100;
   1:  PR[GP1:91,1] = PR[GP1:90,1] + 37.056;
   1:  PR[GP1:91,2] = PR[GP1:90,2] + -34.531;
   1:L PR[91] R[100]mm/sec CNT100;
   1:  PR[GP1:91,1] = PR[GP1:90,1] + 45.579;
   1:  PR[GP1:91,2] = PR[GP1:90,2] + -33.833;
   1:L PR[91] R[100]mm/sec CNT100;
   1:  PR[GP1:91,1] = PR[GP1:90,1] + 48.130;
   1:  PR[GP1:91,2] = PR[GP1:90,2] + -33.445;
   1:L PR[91] R[100]mm/sec CNT100;
   1:  PR[GP1:91,1] = PR[GP1:90,1] + 57.018;
   1:  PR[GP1:91,2] = PR[GP1:90,2] + -29.583;
   1:L PR[91] R[100]mm/sec CNT100;
   1:  PR[GP1:91,1] = PR[GP1:90,1] + 58.405;
   1:  PR[GP1:91,2] = PR[GP1:90,2] + -28.892;
   1:L PR[91] R[100]mm/sec CNT100;
   1:  PR[GP1:91,1] = PR[GP1:90,1] + 66.161;
   1:  PR[GP1:91,2] = PR[GP1:90,2] + -21.815;
   1:L PR[91] R[100]mm/sec CNT100;
   1:  PR[GP1:91,1] = PR[GP1:90,1] + 66.740;
   1:  PR[GP1:91,2] = PR[GP1:90,2] + -21.244;
   1:L PR[91] R[100]mm/sec CNT100;
   1:  PR[GP1:91,1] = PR[GP1:90,1] + 71.999;
   1:  PR[GP1:91,2] = PR[GP1:90,2] + -11.621;
   1:L PR[91] R[100]mm/sec CNT100;
   1:  PR[GP1:91,1] = PR[GP1:90,1] + 72.173;
   1:  PR[GP1:91,2] = PR[GP1:90,2] + -11.284;
   1:L PR[91] R[100]mm/sec CNT100;
   1:  PR[GP1:91,1] = PR[GP1:90,1] + 74.070;
   1:  PR[GP1:91,2] = PR[GP1:90,2] + -0.072;
   1:L PR[91] R[100]mm/sec CNT100;
   1:  PR[GP1:91,1] = PR[GP1:90,1] + 72.173;
   1:  PR[GP1:91,2] = PR[GP1:90,2] + 11.140;
   1:L PR[91] R[100]mm/sec CNT100;
   1:  PR[GP1:91,1] = PR[GP1:90,1] + 71.999;
   1:  PR[GP1:91,2] = PR[GP1:90,2] + 11.477;
   1:L PR[91] R[100]mm/sec CNT100;
   1:  PR[GP1:91,1] = PR[GP1:90,1] + 66.740;
   1:  PR[GP1:91,2] = PR[GP1:90,2] + 21.100;
   1:L PR[91] R[100]mm/sec CNT100;
   1:  PR[GP1:91,1] = PR[GP1:90,1] + 66.161;
   1:  PR[GP1:91,2] = PR[GP1:90,2] + 21.671;
   1:L PR[91] R[100]mm/sec CNT100;
   1:  PR[GP1:91,1] = PR[GP1:90,1] + 58.405;
   1:  PR[GP1:91,2] = PR[GP1:90,2] + 28.748;
   1:L PR[91] R[100]mm/sec CNT100;
   1:  PR[GP1:91,1] = PR[GP1:90,1] + 57.018;
   1:  PR[GP1:91,2] = PR[GP1:90,2] + 29.439;
   1:L PR[91] R[100]mm/sec CNT100;
   1:  PR[GP1:91,1] = PR[GP1:90,1] + 48.130;
   1:  PR[GP1:91,2] = PR[GP1:90,2] + 33.301;
   1:L PR[91] R[100]mm/sec CNT100;
   1:  PR[GP1:91,1] = PR[GP1:90,1] + 45.579;
   1:  PR[GP1:91,2] = PR[GP1:90,2] + 33.689;
   1:L PR[91] R[100]mm/sec CNT100;
   1:  PR[GP1:91,1] = PR[GP1:90,1] + 37.056;
   1:  PR[GP1:91,2] = PR[GP1:90,2] + 34.387;
   1:L PR[91] R[100]mm/sec CNT100;
   1:  PR[GP1:91,1] = PR[GP1:90,1] + 33.266;
   1:  PR[GP1:91,2] = PR[GP1:90,2] + 33.771;
   1:L PR[91] R[100]mm/sec CNT100;
   1:  PR[GP1:91,1] = PR[GP1:90,1] + 26.331;
   1:  PR[GP1:91,2] = PR[GP1:90,2] + 32.026;
   1:L PR[91] R[100]mm/sec CNT100;
   1:  PR[GP1:91,1] = PR[GP1:90,1] + 21.705;
   1:  PR[GP1:91,2] = PR[GP1:90,2] + 29.660;
   1:L PR[91] R[100]mm/sec CNT100;
   1:  PR[GP1:91,1] = PR[GP1:90,1] + 16.971;
   1:  PR[GP1:91,2] = PR[GP1:90,2] + 26.586;
   1:L PR[91] R[100]mm/sec CNT100;
   1:  PR[GP1:91,1] = PR[GP1:90,1] + 12.409;
   1:  PR[GP1:91,2] = PR[GP1:90,2] + 21.999;
   1:L PR[91] R[100]mm/sec CNT100;
   1:  PR[GP1:91,1] = PR[GP1:90,1] + 9.779;
   1:  PR[GP1:91,2] = PR[GP1:90,2] + 18.620;
   1:L PR[91] R[100]mm/sec CNT100;
   1:  PR[GP1:91,1] = PR[GP1:90,1] + 6.367;
   1:  PR[GP1:91,2] = PR[GP1:90,2] + 11.808;
   1:L PR[91] R[100]mm/sec CNT100;
   1:  PR[GP1:91,1] = PR[GP1:90,1] + 5.354;
   1:  PR[GP1:91,2] = PR[GP1:90,2] + 8.823;
   1:L PR[91] R[100]mm/sec CNT100;
   1:  PR[GP1:91,1] = PR[GP1:90,1] + 4.794;
   1:  PR[GP1:91,2] = PR[GP1:90,2] + 7.230;
   1:L PR[91] R[100]mm/sec CNT100;
   1:  PR[GP1:91,1] = PR[GP1:90,1] + 3.717;
   1:  PR[GP1:91,2] = PR[GP1:90,2] + 5.924;
   1:L PR[91] R[100]mm/sec CNT100;
   1:  PR[GP1:91,1] = PR[GP1:90,1] + 2.544;
   1:  PR[GP1:91,2] = PR[GP1:90,2] + 4.649;
   1:L PR[91] R[100]mm/sec CNT100;
   1:  PR[GP1:91,1] = PR[GP1:90,1] + 1.943;
   1:  PR[GP1:91,2] = PR[GP1:90,2] + 4.317;
   1:L PR[91] R[100]mm/sec CNT100;
   1:  PR[GP1:91,1] = PR[GP1:90,1] + 0.753;
   1:  PR[GP1:91,2] = PR[GP1:90,2] + 4.329;
   1:L PR[91] R[100]mm/sec CNT100;
   1:  ! -- Layer/Ebene 34 -- !;
   1:  PR[91] = PR[90];
   1:  PR[GP1:91,1] = PR[GP1:90,1] + -2.165;
   1:  PR[GP1:91,2] = PR[GP1:90,2] + 5.067;
   1:  PR[GP1:91,3] = PR[GP1:90,3] + 21.045;
   1:L PR[91] R[100]mm/sec CNT100;
   1:  PR[GP1:91,1] = PR[GP1:90,1] + -2.544;
   1:  PR[GP1:91,2] = PR[GP1:90,2] + 5.332;
   1:L PR[91] R[100]mm/sec CNT100;
   1:  PR[GP1:91,1] = PR[GP1:90,1] + -3.739;
   1:  PR[GP1:91,2] = PR[GP1:90,2] + 6.797;
   1:L PR[91] R[100]mm/sec CNT100;
   1:  PR[GP1:91,1] = PR[GP1:90,1] + -5.103;
   1:  PR[GP1:91,2] = PR[GP1:90,2] + 9.214;
   1:L PR[91] R[100]mm/sec CNT100;
   1:  PR[GP1:91,1] = PR[GP1:90,1] + -5.802;
   1:  PR[GP1:91,2] = PR[GP1:90,2] + 11.270;
   1:L PR[91] R[100]mm/sec CNT100;
   1:  PR[GP1:91,1] = PR[GP1:90,1] + -9.652;
   1:  PR[GP1:91,2] = PR[GP1:90,2] + 18.969;
   1:L PR[91] R[100]mm/sec CNT100;
   1:  PR[GP1:91,1] = PR[GP1:90,1] + -11.681;
   1:  PR[GP1:91,2] = PR[GP1:90,2] + 21.574;
   1:L PR[91] R[100]mm/sec CNT100;
   1:  PR[GP1:91,1] = PR[GP1:90,1] + -16.892;
   1:  PR[GP1:91,2] = PR[GP1:90,2] + 26.800;
   1:L PR[91] R[100]mm/sec CNT100;
   1:  PR[GP1:91,1] = PR[GP1:90,1] + -20.850;
   1:  PR[GP1:91,2] = PR[GP1:90,2] + 29.370;
   1:L PR[91] R[100]mm/sec CNT100;
   1:  PR[GP1:91,1] = PR[GP1:90,1] + -26.254;
   1:  PR[GP1:91,2] = PR[GP1:90,2] + 32.133;
   1:L PR[91] R[100]mm/sec CNT100;
   1:  PR[GP1:91,1] = PR[GP1:90,1] + -32.349;
   1:  PR[GP1:91,2] = PR[GP1:90,2] + 33.666;
   1:L PR[91] R[100]mm/sec CNT100;
   1:  PR[GP1:91,1] = PR[GP1:90,1] + -36.947;
   1:  PR[GP1:91,2] = PR[GP1:90,2] + 34.412;
   1:L PR[91] R[100]mm/sec CNT100;
   1:  PR[GP1:91,1] = PR[GP1:90,1] + -44.671;
   1:  PR[GP1:91,2] = PR[GP1:90,2] + 33.778;
   1:L PR[91] R[100]mm/sec CNT100;
   1:  PR[GP1:91,1] = PR[GP1:90,1] + -47.974;
   1:  PR[GP1:91,2] = PR[GP1:90,2] + 33.277;
   1:L PR[91] R[100]mm/sec CNT100;
   1:  PR[GP1:91,1] = PR[GP1:90,1] + -56.183;
   1:  PR[GP1:91,2] = PR[GP1:90,2] + 29.708;
   1:L PR[91] R[100]mm/sec CNT100;
   1:  PR[GP1:91,1] = PR[GP1:90,1] + -58.201;
   1:  PR[GP1:91,2] = PR[GP1:90,2] + 28.700;
   1:L PR[91] R[100]mm/sec CNT100;
   1:  PR[GP1:91,1] = PR[GP1:90,1] + -65.449;
   1:  PR[GP1:91,2] = PR[GP1:90,2] + 22.090;
   1:L PR[91] R[100]mm/sec CNT100;
   1:  PR[GP1:91,1] = PR[GP1:90,1] + -66.497;
   1:  PR[GP1:91,2] = PR[GP1:90,2] + 21.059;
   1:L PR[91] R[100]mm/sec CNT100;
   1:  PR[GP1:91,1] = PR[GP1:90,1] + -71.446;
   1:  PR[GP1:91,2] = PR[GP1:90,2] + 11.996;
   1:L PR[91] R[100]mm/sec CNT100;
   1:  PR[GP1:91,1] = PR[GP1:90,1] + -71.903;
   1:  PR[GP1:91,2] = PR[GP1:90,2] + 11.110;
   1:L PR[91] R[100]mm/sec CNT100;
   1:  PR[GP1:91,1] = PR[GP1:90,1] + -73.791;
   1:  PR[GP1:91,2] = PR[GP1:90,2] + -0.072;
   1:L PR[91] R[100]mm/sec CNT100;
   1:  PR[GP1:91,1] = PR[GP1:90,1] + -72.047;
   1:  PR[GP1:91,2] = PR[GP1:90,2] + -10.354;
   1:L PR[91] R[100]mm/sec CNT100;
   1:  PR[GP1:91,1] = PR[GP1:90,1] + -71.902;
   1:  PR[GP1:91,2] = PR[GP1:90,2] + -11.256;
   1:L PR[91] R[100]mm/sec CNT100;
   1:  PR[GP1:91,1] = PR[GP1:90,1] + -71.446;
   1:  PR[GP1:91,2] = PR[GP1:90,2] + -12.140;
   1:L PR[91] R[100]mm/sec CNT100;
   1:  PR[GP1:91,1] = PR[GP1:90,1] + -66.497;
   1:  PR[GP1:91,2] = PR[GP1:90,2] + -21.203;
   1:L PR[91] R[100]mm/sec CNT100;
   1:  PR[GP1:91,1] = PR[GP1:90,1] + -65.450;
   1:  PR[GP1:91,2] = PR[GP1:90,2] + -22.234;
   1:L PR[91] R[100]mm/sec CNT100;
   1:  PR[GP1:91,1] = PR[GP1:90,1] + -58.201;
   1:  PR[GP1:91,2] = PR[GP1:90,2] + -28.844;
   1:L PR[91] R[100]mm/sec CNT100;
   1:  PR[GP1:91,1] = PR[GP1:90,1] + -56.183;
   1:  PR[GP1:91,2] = PR[GP1:90,2] + -29.852;
   1:L PR[91] R[100]mm/sec CNT100;
   1:  PR[GP1:91,1] = PR[GP1:90,1] + -47.975;
   1:  PR[GP1:91,2] = PR[GP1:90,2] + -33.420;
   1:L PR[91] R[100]mm/sec CNT100;
   1:  PR[GP1:91,1] = PR[GP1:90,1] + -44.671;
   1:  PR[GP1:91,2] = PR[GP1:90,2] + -33.922;
   1:L PR[91] R[100]mm/sec CNT100;
   1:  PR[GP1:91,1] = PR[GP1:90,1] + -36.947;
   1:  PR[GP1:91,2] = PR[GP1:90,2] + -34.556;
   1:L PR[91] R[100]mm/sec CNT100;
   1:  PR[GP1:91,1] = PR[GP1:90,1] + -32.349;
   1:  PR[GP1:91,2] = PR[GP1:90,2] + -33.810;
   1:L PR[91] R[100]mm/sec CNT100;
   1:  PR[GP1:91,1] = PR[GP1:90,1] + -26.254;
   1:  PR[GP1:91,2] = PR[GP1:90,2] + -32.277;
   1:L PR[91] R[100]mm/sec CNT100;
   1:  PR[GP1:91,1] = PR[GP1:90,1] + -20.850;
   1:  PR[GP1:91,2] = PR[GP1:90,2] + -29.514;
   1:L PR[91] R[100]mm/sec CNT100;
   1:  PR[GP1:91,1] = PR[GP1:90,1] + -16.893;
   1:  PR[GP1:91,2] = PR[GP1:90,2] + -26.944;
   1:L PR[91] R[100]mm/sec CNT100;
   1:  PR[GP1:91,1] = PR[GP1:90,1] + -11.681;
   1:  PR[GP1:91,2] = PR[GP1:90,2] + -21.718;
   1:L PR[91] R[100]mm/sec CNT100;
   1:  PR[GP1:91,1] = PR[GP1:90,1] + -9.652;
   1:  PR[GP1:91,2] = PR[GP1:90,2] + -19.113;
   1:L PR[91] R[100]mm/sec CNT100;
   1:  PR[GP1:91,1] = PR[GP1:90,1] + -5.807;
   1:  PR[GP1:91,2] = PR[GP1:90,2] + -11.430;
   1:L PR[91] R[100]mm/sec CNT100;
   1:  PR[GP1:91,1] = PR[GP1:90,1] + -4.619;
   1:  PR[GP1:91,2] = PR[GP1:90,2] + -7.976;
   1:L PR[91] R[100]mm/sec CNT100;
   1:  PR[GP1:91,1] = PR[GP1:90,1] + -3.469;
   1:  PR[GP1:91,2] = PR[GP1:90,2] + -6.705;
   1:L PR[91] R[100]mm/sec CNT100;
   1:  PR[GP1:91,1] = PR[GP1:90,1] + -3.150;
   1:  PR[GP1:91,2] = PR[GP1:90,2] + -6.510;
   1:L PR[91] R[100]mm/sec CNT100;
   1:  PR[GP1:91,1] = PR[GP1:90,1] + -1.873;
   1:  PR[GP1:91,2] = PR[GP1:90,2] + -4.984;
   1:L PR[91] R[100]mm/sec CNT100;
   1:  PR[GP1:91,1] = PR[GP1:90,1] + 1.101;
   1:  PR[GP1:91,2] = PR[GP1:90,2] + -5.213;
   1:L PR[91] R[100]mm/sec CNT100;
   1:  PR[GP1:91,1] = PR[GP1:90,1] + 1.231;
   1:  PR[GP1:91,2] = PR[GP1:90,2] + -5.318;
   1:L PR[91] R[100]mm/sec CNT100;
   1:  PR[GP1:91,1] = PR[GP1:90,1] + 2.676;
   1:  PR[GP1:91,2] = PR[GP1:90,2] + -5.303;
   1:L PR[91] R[100]mm/sec CNT100;
   1:  PR[GP1:91,1] = PR[GP1:90,1] + 3.983;
   1:  PR[GP1:91,2] = PR[GP1:90,2] + -7.790;
   1:L PR[91] R[100]mm/sec CNT100;
   1:  PR[GP1:91,1] = PR[GP1:90,1] + 5.292;
   1:  PR[GP1:91,2] = PR[GP1:90,2] + -9.298;
   1:L PR[91] R[100]mm/sec CNT100;
   1:  PR[GP1:91,1] = PR[GP1:90,1] + 6.015;
   1:  PR[GP1:91,2] = PR[GP1:90,2] + -11.426;
   1:L PR[91] R[100]mm/sec CNT100;
   1:  PR[GP1:91,1] = PR[GP1:90,1] + 9.857;
   1:  PR[GP1:91,2] = PR[GP1:90,2] + -19.094;
   1:L PR[91] R[100]mm/sec CNT100;
   1:  PR[GP1:91,1] = PR[GP1:90,1] + 11.886;
   1:  PR[GP1:91,2] = PR[GP1:90,2] + -21.699;
   1:L PR[91] R[100]mm/sec CNT100;
   1:  PR[GP1:91,1] = PR[GP1:90,1] + 17.098;
   1:  PR[GP1:91,2] = PR[GP1:90,2] + -26.941;
   1:L PR[91] R[100]mm/sec CNT100;
   1:  PR[GP1:91,1] = PR[GP1:90,1] + 21.054;
   1:  PR[GP1:91,2] = PR[GP1:90,2] + -29.510;
   1:L PR[91] R[100]mm/sec CNT100;
   1:  PR[GP1:91,1] = PR[GP1:90,1] + 26.460;
   1:  PR[GP1:91,2] = PR[GP1:90,2] + -32.273;
   1:L PR[91] R[100]mm/sec CNT100;
   1:  PR[GP1:91,1] = PR[GP1:90,1] + 32.555;
   1:  PR[GP1:91,2] = PR[GP1:90,2] + -33.807;
   1:L PR[91] R[100]mm/sec CNT100;
   1:  PR[GP1:91,1] = PR[GP1:90,1] + 37.155;
   1:  PR[GP1:91,2] = PR[GP1:90,2] + -34.556;
   1:L PR[91] R[100]mm/sec CNT100;
   1:  PR[GP1:91,1] = PR[GP1:90,1] + 44.879;
   1:  PR[GP1:91,2] = PR[GP1:90,2] + -33.922;
   1:L PR[91] R[100]mm/sec CNT100;
   1:  PR[GP1:91,1] = PR[GP1:90,1] + 48.184;
   1:  PR[GP1:91,2] = PR[GP1:90,2] + -33.421;
   1:L PR[91] R[100]mm/sec CNT100;
   1:  PR[GP1:91,1] = PR[GP1:90,1] + 56.394;
   1:  PR[GP1:91,2] = PR[GP1:90,2] + -29.854;
   1:L PR[91] R[100]mm/sec CNT100;
   1:  PR[GP1:91,1] = PR[GP1:90,1] + 58.413;
   1:  PR[GP1:91,2] = PR[GP1:90,2] + -28.847;
   1:L PR[91] R[100]mm/sec CNT100;
   1:  PR[GP1:91,1] = PR[GP1:90,1] + 65.661;
   1:  PR[GP1:91,2] = PR[GP1:90,2] + -22.233;
   1:L PR[91] R[100]mm/sec CNT100;
   1:  PR[GP1:91,1] = PR[GP1:90,1] + 66.709;
   1:  PR[GP1:91,2] = PR[GP1:90,2] + -21.201;
   1:L PR[91] R[100]mm/sec CNT100;
   1:  PR[GP1:91,1] = PR[GP1:90,1] + 71.659;
   1:  PR[GP1:91,2] = PR[GP1:90,2] + -12.143;
   1:L PR[91] R[100]mm/sec CNT100;
   1:  PR[GP1:91,1] = PR[GP1:90,1] + 72.116;
   1:  PR[GP1:91,2] = PR[GP1:90,2] + -11.260;
   1:L PR[91] R[100]mm/sec CNT100;
   1:  PR[GP1:91,1] = PR[GP1:90,1] + 74.004;
   1:  PR[GP1:91,2] = PR[GP1:90,2] + -0.072;
   1:L PR[91] R[100]mm/sec CNT100;
   1:  PR[GP1:91,1] = PR[GP1:90,1] + 72.116;
   1:  PR[GP1:91,2] = PR[GP1:90,2] + 11.116;
   1:L PR[91] R[100]mm/sec CNT100;
   1:  PR[GP1:91,1] = PR[GP1:90,1] + 71.659;
   1:  PR[GP1:91,2] = PR[GP1:90,2] + 11.999;
   1:L PR[91] R[100]mm/sec CNT100;
   1:  PR[GP1:91,1] = PR[GP1:90,1] + 66.709;
   1:  PR[GP1:91,2] = PR[GP1:90,2] + 21.057;
   1:L PR[91] R[100]mm/sec CNT100;
   1:  PR[GP1:91,1] = PR[GP1:90,1] + 65.661;
   1:  PR[GP1:91,2] = PR[GP1:90,2] + 22.089;
   1:L PR[91] R[100]mm/sec CNT100;
   1:  PR[GP1:91,1] = PR[GP1:90,1] + 58.413;
   1:  PR[GP1:91,2] = PR[GP1:90,2] + 28.703;
   1:L PR[91] R[100]mm/sec CNT100;
   1:  PR[GP1:91,1] = PR[GP1:90,1] + 56.394;
   1:  PR[GP1:91,2] = PR[GP1:90,2] + 29.710;
   1:L PR[91] R[100]mm/sec CNT100;
   1:  PR[GP1:91,1] = PR[GP1:90,1] + 48.184;
   1:  PR[GP1:91,2] = PR[GP1:90,2] + 33.277;
   1:L PR[91] R[100]mm/sec CNT100;
   1:  PR[GP1:91,1] = PR[GP1:90,1] + 44.879;
   1:  PR[GP1:91,2] = PR[GP1:90,2] + 33.778;
   1:L PR[91] R[100]mm/sec CNT100;
   1:  PR[GP1:91,1] = PR[GP1:90,1] + 37.155;
   1:  PR[GP1:91,2] = PR[GP1:90,2] + 34.412;
   1:L PR[91] R[100]mm/sec CNT100;
   1:  PR[GP1:91,1] = PR[GP1:90,1] + 32.555;
   1:  PR[GP1:91,2] = PR[GP1:90,2] + 33.663;
   1:L PR[91] R[100]mm/sec CNT100;
   1:  PR[GP1:91,1] = PR[GP1:90,1] + 26.460;
   1:  PR[GP1:91,2] = PR[GP1:90,2] + 32.129;
   1:L PR[91] R[100]mm/sec CNT100;
   1:  PR[GP1:91,1] = PR[GP1:90,1] + 21.054;
   1:  PR[GP1:91,2] = PR[GP1:90,2] + 29.366;
   1:L PR[91] R[100]mm/sec CNT100;
   1:  PR[GP1:91,1] = PR[GP1:90,1] + 17.098;
   1:  PR[GP1:91,2] = PR[GP1:90,2] + 26.797;
   1:L PR[91] R[100]mm/sec CNT100;
   1:  PR[GP1:91,1] = PR[GP1:90,1] + 11.886;
   1:  PR[GP1:91,2] = PR[GP1:90,2] + 21.555;
   1:L PR[91] R[100]mm/sec CNT100;
   1:  PR[GP1:91,1] = PR[GP1:90,1] + 9.857;
   1:  PR[GP1:91,2] = PR[GP1:90,2] + 18.950;
   1:L PR[91] R[100]mm/sec CNT100;
   1:  PR[GP1:91,1] = PR[GP1:90,1] + 6.008;
   1:  PR[GP1:91,2] = PR[GP1:90,2] + 11.264;
   1:L PR[91] R[100]mm/sec CNT100;
   1:  PR[GP1:91,1] = PR[GP1:90,1] + 4.828;
   1:  PR[GP1:91,2] = PR[GP1:90,2] + 7.829;
   1:L PR[91] R[100]mm/sec CNT100;
   1:  PR[GP1:91,1] = PR[GP1:90,1] + 3.593;
   1:  PR[GP1:91,2] = PR[GP1:90,2] + 6.333;
   1:L PR[91] R[100]mm/sec CNT100;
   1:  PR[GP1:91,1] = PR[GP1:90,1] + 2.516;
   1:  PR[GP1:91,2] = PR[GP1:90,2] + 5.162;
   1:L PR[91] R[100]mm/sec CNT100;
   1:  PR[GP1:91,1] = PR[GP1:90,1] + 1.948;
   1:  PR[GP1:91,2] = PR[GP1:90,2] + 4.848;
   1:L PR[91] R[100]mm/sec CNT100;
   1:  PR[GP1:91,1] = PR[GP1:90,1] + 0.536;
   1:  PR[GP1:91,2] = PR[GP1:90,2] + 4.862;
   1:L PR[91] R[100]mm/sec CNT100;
   1:  ! -- Layer/Ebene 35 -- !;
   1:  PR[91] = PR[90];
   1:  PR[GP1:91,1] = PR[GP1:90,1] + -2.142;
   1:  PR[GP1:91,2] = PR[GP1:90,2] + 5.582;
   1:  PR[GP1:91,3] = PR[GP1:90,3] + 21.655;
   1:L PR[91] R[100]mm/sec CNT100;
   1:  PR[GP1:91,1] = PR[GP1:90,1] + -2.504;
   1:  PR[GP1:91,2] = PR[GP1:90,2] + 5.836;
   1:L PR[91] R[100]mm/sec CNT100;
   1:  PR[GP1:91,1] = PR[GP1:90,1] + -3.885;
   1:  PR[GP1:91,2] = PR[GP1:90,2] + 7.528;
   1:L PR[91] R[100]mm/sec CNT100;
   1:  PR[GP1:91,1] = PR[GP1:90,1] + -5.079;
   1:  PR[GP1:91,2] = PR[GP1:90,2] + 9.655;
   1:L PR[91] R[100]mm/sec CNT100;
   1:  PR[GP1:91,1] = PR[GP1:90,1] + -5.444;
   1:  PR[GP1:91,2] = PR[GP1:90,2] + 10.727;
   1:L PR[91] R[100]mm/sec CNT100;
   1:  PR[GP1:91,1] = PR[GP1:90,1] + -9.731;
   1:  PR[GP1:91,2] = PR[GP1:90,2] + 19.301;
   1:L PR[91] R[100]mm/sec CNT100;
   1:  PR[GP1:91,1] = PR[GP1:90,1] + -11.158;
   1:  PR[GP1:91,2] = PR[GP1:90,2] + 21.132;
   1:L PR[91] R[100]mm/sec CNT100;
   1:  PR[GP1:91,1] = PR[GP1:90,1] + -17.020;
   1:  PR[GP1:91,2] = PR[GP1:90,2] + 27.011;
   1:L PR[91] R[100]mm/sec CNT100;
   1:  PR[GP1:91,1] = PR[GP1:90,1] + -20.200;
   1:  PR[GP1:91,2] = PR[GP1:90,2] + 29.076;
   1:L PR[91] R[100]mm/sec CNT100;
   1:  PR[GP1:91,1] = PR[GP1:90,1] + -26.383;
   1:  PR[GP1:91,2] = PR[GP1:90,2] + 32.237;
   1:L PR[91] R[100]mm/sec CNT100;
   1:  PR[GP1:91,1] = PR[GP1:90,1] + -31.639;
   1:  PR[GP1:91,2] = PR[GP1:90,2] + 33.559;
   1:L PR[91] R[100]mm/sec CNT100;
   1:  PR[GP1:91,1] = PR[GP1:90,1] + -37.046;
   1:  PR[GP1:91,2] = PR[GP1:90,2] + 34.436;
   1:L PR[91] R[100]mm/sec CNT100;
   1:  PR[GP1:91,1] = PR[GP1:90,1] + -43.973;
   1:  PR[GP1:91,2] = PR[GP1:90,2] + 33.868;
   1:L PR[91] R[100]mm/sec CNT100;
   1:  PR[GP1:91,1] = PR[GP1:90,1] + -48.029;
   1:  PR[GP1:91,2] = PR[GP1:90,2] + 33.252;
   1:L PR[91] R[100]mm/sec CNT100;
   1:  PR[GP1:91,1] = PR[GP1:90,1] + -55.560;
   1:  PR[GP1:91,2] = PR[GP1:90,2] + 29.978;
   1:L PR[91] R[100]mm/sec CNT100;
   1:  PR[GP1:91,1] = PR[GP1:90,1] + -58.209;
   1:  PR[GP1:91,2] = PR[GP1:90,2] + 28.655;
   1:L PR[91] R[100]mm/sec CNT100;
   1:  PR[GP1:91,1] = PR[GP1:90,1] + -64.950;
   1:  PR[GP1:91,2] = PR[GP1:90,2] + 22.507;
   1:L PR[91] R[100]mm/sec CNT100;
   1:  PR[GP1:91,1] = PR[GP1:90,1] + -66.466;
   1:  PR[GP1:91,2] = PR[GP1:90,2] + 21.016;
   1:L PR[91] R[100]mm/sec CNT100;
   1:  PR[GP1:91,1] = PR[GP1:90,1] + -71.106;
   1:  PR[GP1:91,2] = PR[GP1:90,2] + 12.518;
   1:L PR[91] R[100]mm/sec CNT100;
   1:  PR[GP1:91,1] = PR[GP1:90,1] + -71.846;
   1:  PR[GP1:91,2] = PR[GP1:90,2] + 11.085;
   1:L PR[91] R[100]mm/sec CNT100;
   1:  PR[GP1:91,1] = PR[GP1:90,1] + -73.724;
   1:  PR[GP1:91,2] = PR[GP1:90,2] + -0.072;
   1:L PR[91] R[100]mm/sec CNT100;
   1:  PR[GP1:91,1] = PR[GP1:90,1] + -72.079;
   1:  PR[GP1:91,2] = PR[GP1:90,2] + -9.768;
   1:L PR[91] R[100]mm/sec CNT100;
   1:  PR[GP1:91,1] = PR[GP1:90,1] + -71.845;
   1:  PR[GP1:91,2] = PR[GP1:90,2] + -11.231;
   1:L PR[91] R[100]mm/sec CNT100;
   1:  PR[GP1:91,1] = PR[GP1:90,1] + -71.106;
   1:  PR[GP1:91,2] = PR[GP1:90,2] + -12.662;
   1:L PR[91] R[100]mm/sec CNT100;
   1:  PR[GP1:91,1] = PR[GP1:90,1] + -66.466;
   1:  PR[GP1:91,2] = PR[GP1:90,2] + -21.160;
   1:L PR[91] R[100]mm/sec CNT100;
   1:  PR[GP1:91,1] = PR[GP1:90,1] + -64.950;
   1:  PR[GP1:91,2] = PR[GP1:90,2] + -22.651;
   1:L PR[91] R[100]mm/sec CNT100;
   1:  PR[GP1:91,1] = PR[GP1:90,1] + -58.209;
   1:  PR[GP1:91,2] = PR[GP1:90,2] + -28.799;
   1:L PR[91] R[100]mm/sec CNT100;
   1:  PR[GP1:91,1] = PR[GP1:90,1] + -55.560;
   1:  PR[GP1:91,2] = PR[GP1:90,2] + -30.122;
   1:L PR[91] R[100]mm/sec CNT100;
   1:  PR[GP1:91,1] = PR[GP1:90,1] + -48.029;
   1:  PR[GP1:91,2] = PR[GP1:90,2] + -33.396;
   1:L PR[91] R[100]mm/sec CNT100;
   1:  PR[GP1:91,1] = PR[GP1:90,1] + -43.973;
   1:  PR[GP1:91,2] = PR[GP1:90,2] + -34.012;
   1:L PR[91] R[100]mm/sec CNT100;
   1:  PR[GP1:91,1] = PR[GP1:90,1] + -37.046;
   1:  PR[GP1:91,2] = PR[GP1:90,2] + -34.580;
   1:L PR[91] R[100]mm/sec CNT100;
   1:  PR[GP1:91,1] = PR[GP1:90,1] + -31.639;
   1:  PR[GP1:91,2] = PR[GP1:90,2] + -33.703;
   1:L PR[91] R[100]mm/sec CNT100;
   1:  PR[GP1:91,1] = PR[GP1:90,1] + -26.383;
   1:  PR[GP1:91,2] = PR[GP1:90,2] + -32.381;
   1:L PR[91] R[100]mm/sec CNT100;
   1:  PR[GP1:91,1] = PR[GP1:90,1] + -20.200;
   1:  PR[GP1:91,2] = PR[GP1:90,2] + -29.220;
   1:L PR[91] R[100]mm/sec CNT100;
   1:  PR[GP1:91,1] = PR[GP1:90,1] + -17.020;
   1:  PR[GP1:91,2] = PR[GP1:90,2] + -27.155;
   1:L PR[91] R[100]mm/sec CNT100;
   1:  PR[GP1:91,1] = PR[GP1:90,1] + -11.158;
   1:  PR[GP1:91,2] = PR[GP1:90,2] + -21.276;
